// TIA Portal V16 export
// export: Created 2021-11-12T13:31:33.7596207Z, ExportSetting WithDefaults, DisplayName Totally Integrated Automation Portal, DisplayVersion V16 Update 3, DisplayName TIA Portal Version Control Interface, DisplayVersion V16 Update 2, DisplayName TIA Portal Openness, DisplayVersion V16 Update 3, DisplayName SINAMICS Startdrive Advanced, DisplayVersion V16 Update 5, DisplayName SINAMICS Startdrive G130, G150, S120, S150, SINAMICS MV, S210, DisplayVersion V16 Update 5, DisplayName SINAMICS Startdrive G110M, G120, G120C, G120D, G120P, G115D, DisplayVersion V16 Update 5, DisplayName STEP 7 Professional, DisplayVersion V16 Update 3, DisplayName STEP 7 Safety, DisplayVersion V16, DisplayName WinCC UA Professional, DisplayVersion V16 Update 3
FUNCTION_BLOCK "STD_Siemens_G120_CU240E_2_PN"   // FB1999, LAD
TITLE = Sinamics G120 with CU240E-2 PN control
{ S7_Optimized_Access := 'TRUE' }
AUTHOR : PI
FAMILY : Standard
VERSION : 0.1
// Control of Sinamics G120 with CU240E-2 PN
// 7words in/6words out (to/from PLC)
// Bi directional
// Speed and ramp control
// Errors of FI and motor evaluation
// stored: AutoNumber true, IsIECCheckEnabled false, IsRetainMemResEnabled false, MemoryReserve 100, SetENOAutomatically false, UDAEnableTagReadback false
   VAR_INPUT
      IW_HWID : HW_SUBMODULE;   // HW_Identifier - for read and write
      IB1ReqDir1 : Bool;   // Request to move in direction 1
      IB1ReqDir2 : Bool;   // Request to move in direction 2
      IB1Ack : Bool;   // Acknowledge
      IB1AlmSupp : Bool;   // Alarm suppression - external
      IB1FIProt : Bool;   // Alarm: FI Circuit Breaker / Protection of Frequency inverter OK
      IB1FICont : Bool;   // Alarm: FI Contactor / Signal from contactor on FIs input
      IB1MtrServSwch : Bool;   // Alarm: Motor 1 Service Switch / Service switch in front of motor
      IB1MtrTemp : Bool;   // Alarm: Motor 1 Thermal Protection / Temperature of motor OK
      IB1MtrBrkProt : Bool;   // Alarm: Motor 1 Brake Circuit Breaker / Protection of brake OK
      IB1MtrBrkCont : Bool;   // Alarm: Motor 1 Brake Contactor / Contactor of brake
      IB0OFF2 : Bool;   // Signal to activate OFF2 (coast)
      IB0OFF3 : Bool;   // Signal to activate OFF3 (fast ramp)
      IR_SpdSP : Real;   // Requested speed (rpm)
      IR_UpRamp { ExternalAccessible := 'False'; ExternalVisible := 'False'; ExternalWritable := 'False'} : Real := 100.0;   // Up ramp scaling 0..100%
      IR_DownRamp { ExternalAccessible := 'False'; ExternalVisible := 'False'; ExternalWritable := 'False'} : Real := 100.0;   // Down ramp scaling 0..100%
      IT_FIAlmFbk { ExternalAccessible := 'False'; ExternalVisible := 'False'; ExternalWritable := 'False'} : Time := T#100ms;   // Time to evaluate error of FI feedback
      IT_BrkAlm : Time;   // Time to evaluate error of brake release feedback
      IT_Rot : Time := T#100ms;   // Timeout for sense of rotation evaluation
   END_VAR
   VAR_OUTPUT
      OS_Status : Struct   // Output structures
         Main : "UDT_Status_main";
         Specific : "UDT_SINAMICS_G120_Status_specific";
         Error : "UDT_Error02";
      END_STRUCT;
      OW_CtrlWord1 : Word;   // Control word to FI -just for monitoring
      OB1_MtrHoldBrkOpn : Bool;   // Motor holding brake open
   END_VAR
   VAR_IN_OUT
      XS_Command : "UDT_SINAMICS_G120_Command";
      XS_Parameter : "UDT_SINAMICS_G120_Parameter";
   END_VAR
   VAR DB_SPECIFIC
      SS_Alarm : Struct   // Alarms
         FIProt : Bool;   // Frekvenční měnič - ochrana / Frequency invertor - protection / Convertisseur de fréquence - protection
         FICont : Bool;   // Frekvenční měnič - spínač / Frequency invertor - contactor / Convertisseur de fréquence - contacteur
         FIFastOff : Bool;   // Frekvenční měnič - porucha / Frequency invertor - fast off / Convertisseur de fréquence - erreur
         FIFbk : Bool;   // Frekvenční měnič - zpětná vazba chod / Frequency invertor - feedback run / Convertisseur de fréquence - rétroaction
         FITemp : Bool;   // Frekvenční měnič - vysoká teplota / Frequency invertor - high temperature / Convertisseur de fréquence - température
         FICommErr : Bool;   // Frekvenční měnič - komunikace / Frequency invertor - communication / Convertisseur de fréquence - communication
         FINotRdy : Bool;   // Frequency invertor - not ready
         Res_0_7 : Bool;   // Reserve
         MtrServSwch : Bool;   // Motor - servisní vypínač / Motor - service switch / Moteur - interrupteur de service
         MtrTemp : Bool;   // Motor - vysoká teplota / Motor - high temperature / Moteur - température
         MtrBrkProt : Bool;   // Motor - ochrana brzdy / Motor - brake protection / Moteur - protectrice de frein
         MtrBrkCont : Bool;   // Motor - spínač brzdy / Motor - brake contactor / Moteur - contacteur de frein
         MtrRot : Bool;   // Motor - sense of rotation incoherence
         Res_1_5 : Bool;   // Reserve
         Res_1_6 : Bool;   // Reserve
         InCmdIncoher : Bool;   // Dir1 and Dir2 input commands incoherence
      END_STRUCT;
      SS_Warning : Struct   // Warnings
         SpdDeviation : Bool;   // Speed deviation outside the tolerance range
         Res_0_1 : Bool;   // Reserve
         Res_0_2 : Bool;   // Reserve
         Res_0_3 : Bool;   // Reserve
         Res_0_4 : Bool;   // Reserve
         Res_0_5 : Bool;   // Reserve
         Res_0_6 : Bool;   // Reserve
         Res_0_7 : Bool;   // Reserve
         Res_1_0 : Bool;   // Reserve
         Res_1_1 : Bool;   // Reserve
         Res_1_2 : Bool;   // Reserve
         Res_1_3 : Bool;   // Reserve
         Res_1_4 : Bool;   // Reserve
         Res_1_5 : Bool;   // Reserve
         Res_1_6 : Bool;   // Reserve
         Res_1_7 : Bool;   // Reserve
      END_STRUCT;
      SI_DPRDDATRetVal { ExternalAccessible := 'False'; ExternalVisible := 'False'; ExternalWritable := 'False'} : Int;   // DPRD_DAT function return value
      SI_DPWRDATRetVal { ExternalAccessible := 'False'; ExternalVisible := 'False'; ExternalWritable := 'False'} : Int;   // DPWR_DAT function return value
      SB1DPRDWRCommOK : Bool;   // No error occurs while the instruction DPRD_DAT or DPWR_DAT is being executed
      SB1OutDir1 : Bool;   // Request to move in direction 1
      SB1OutDir2 : Bool;   // Request to move in direction 2
      ST_AlmFbk { S7_SetPoint := 'True'} : TON_TIME;   // To evaluate feedback error of FI
      ST_AlmBrake { S7_SetPoint := 'True'} : TON_TIME;   // To evaluate error on brake
      ST_AlmFIErr { S7_SetPoint := 'True'} : TON_TIME;   // To evaluate error reported from FI
   END_VAR
   VAR
      ST_RotSense { S7_SetPoint := 'True'} : TON_TIME;   // To evaluate sense of rotation incoherence
   END_VAR
   VAR DB_SPECIFIC
      ST_AckFl { S7_SetPoint := 'True'} : TP_TIME;   // TOF ack to G120
   END_VAR
   VAR_TEMP
      TS_Command : "UDT_SINAMICS_G120_Command";
      TS_Parameter : "UDT_SINAMICS_G120_Parameter";
      TS_Status : Struct
         Main : "UDT_Status_main";
         Specific : "UDT_SINAMICS_G120_Status_specific";
         Error : "UDT_Error02";
      END_STRUCT;
      TI_DPReadRet : Int;   // Result of DP reading
      TI_DPWriteRet : Int;   // Result of DP writing
      TR_Temp : Real;   // Temporary REAL value
      TS_Input : "UDT_ CU240E_I_352";   // 6 byte struct to receive data from FI
      TS_Output : "UDT_CU240E_O_352";   // 6 byte struct to send data to FI
   END_VAR
   VAR CONSTANT
      Ack : Time := T#300ms;   // Time to acknowledge FI (via PN)
   END_VAR
BEGIN

REGION Network 1: Clear temporary variables, TS_Status - Main, Specific
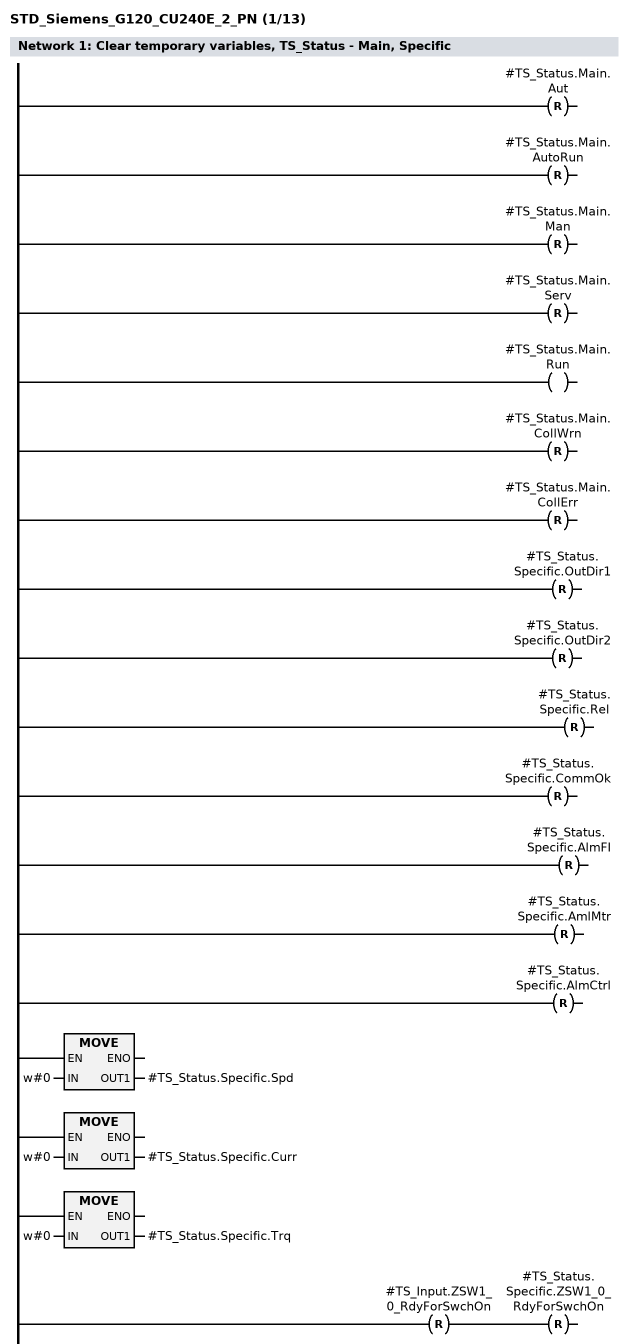
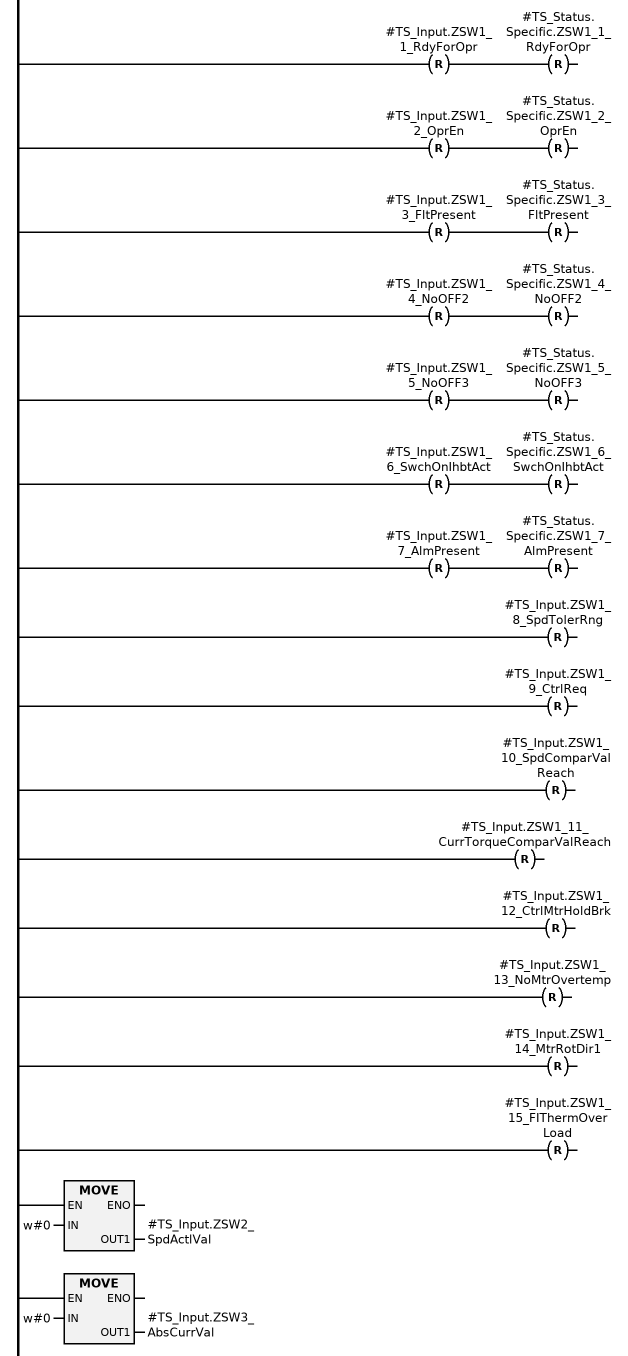
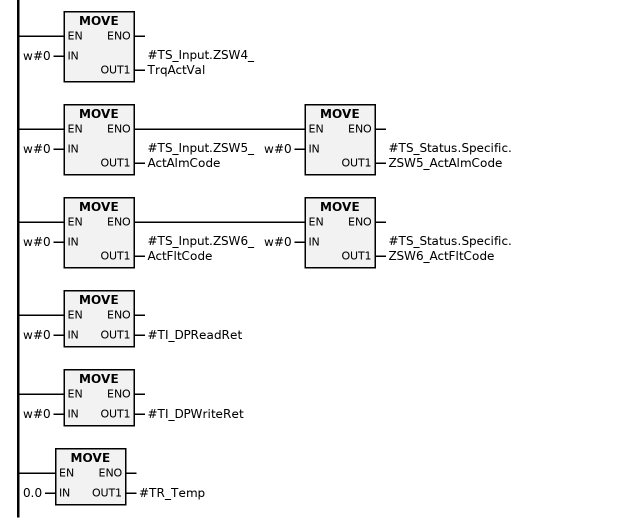
   RUNG wire#powerrail
      R_Coil( #TS_Status.Main.Aut )
   END_RUNG
   RUNG wire#powerrail
      R_Coil( #TS_Status.Main.AutoRun )
   END_RUNG
   RUNG wire#powerrail
      R_Coil( #TS_Status.Main.Man )
   END_RUNG
   RUNG wire#powerrail
      R_Coil( #TS_Status.Main.Serv )
   END_RUNG
   RUNG wire#powerrail
      Coil( #TS_Status.Main.Run )
   END_RUNG
   RUNG wire#powerrail
      R_Coil( #TS_Status.Main.CollWrn )
   END_RUNG
   RUNG wire#powerrail
      R_Coil( #TS_Status.Main.CollErr )
   END_RUNG
   RUNG wire#powerrail
      R_Coil( #TS_Status.Specific.OutDir1 )
   END_RUNG
   RUNG wire#powerrail
      R_Coil( #TS_Status.Specific.OutDir2 )
   END_RUNG
   RUNG wire#powerrail
      R_Coil( #TS_Status.Specific.Rel )
   END_RUNG
   RUNG wire#powerrail
      R_Coil( #TS_Status.Specific.CommOk )
   END_RUNG
   RUNG wire#powerrail
      R_Coil( #TS_Status.Specific.AlmFI )
   END_RUNG
   RUNG wire#powerrail
      R_Coil( #TS_Status.Specific.AmlMtr )
   END_RUNG
   RUNG wire#powerrail
      R_Coil( #TS_Status.Specific.AlmCtrl )
   END_RUNG
   RUNG wire#powerrail
      { S7_GenerateENO := "TRUE" } Move(in := w#0, out1 => #TS_Status.Specific.Spd)
   END_RUNG
   RUNG wire#powerrail
      { S7_GenerateENO := "TRUE" } Move(in := w#0, out1 => #TS_Status.Specific.Curr)
   END_RUNG
   RUNG wire#powerrail
      { S7_GenerateENO := "TRUE" } Move(in := w#0, out1 => #TS_Status.Specific.Trq)
   END_RUNG
   RUNG wire#powerrail
      R_Coil( #TS_Input.ZSW1_0_RdyForSwchOn )
      R_Coil( #TS_Status.Specific.ZSW1_0_RdyForSwchOn )
   END_RUNG
   RUNG wire#powerrail
      R_Coil( #TS_Input.ZSW1_1_RdyForOpr )
      R_Coil( #TS_Status.Specific.ZSW1_1_RdyForOpr )
   END_RUNG
   RUNG wire#powerrail
      R_Coil( #TS_Input.ZSW1_2_OprEn )
      R_Coil( #TS_Status.Specific.ZSW1_2_OprEn )
   END_RUNG
   RUNG wire#powerrail
      R_Coil( #TS_Input.ZSW1_3_FltPresent )
      R_Coil( #TS_Status.Specific.ZSW1_3_FltPresent )
   END_RUNG
   RUNG wire#powerrail
      R_Coil( #TS_Input.ZSW1_4_NoOFF2 )
      R_Coil( #TS_Status.Specific.ZSW1_4_NoOFF2 )
   END_RUNG
   RUNG wire#powerrail
      R_Coil( #TS_Input.ZSW1_5_NoOFF3 )
      R_Coil( #TS_Status.Specific.ZSW1_5_NoOFF3 )
   END_RUNG
   RUNG wire#powerrail
      R_Coil( #TS_Input.ZSW1_6_SwchOnIhbtAct )
      R_Coil( #TS_Status.Specific.ZSW1_6_SwchOnIhbtAct )
   END_RUNG
   RUNG wire#powerrail
      R_Coil( #TS_Input.ZSW1_7_AlmPresent )
      R_Coil( #TS_Status.Specific.ZSW1_7_AlmPresent )
   END_RUNG
   RUNG wire#powerrail
      R_Coil( #TS_Input.ZSW1_8_SpdTolerRng )
   END_RUNG
   RUNG wire#powerrail
      R_Coil( #TS_Input.ZSW1_9_CtrlReq )
   END_RUNG
   RUNG wire#powerrail
      R_Coil( #TS_Input.ZSW1_10_SpdComparValReach )
   END_RUNG
   RUNG wire#powerrail
      R_Coil( #TS_Input.ZSW1_11_CurrTorqueComparValReach )
   END_RUNG
   RUNG wire#powerrail
      R_Coil( #TS_Input.ZSW1_12_CtrlMtrHoldBrk )
   END_RUNG
   RUNG wire#powerrail
      R_Coil( #TS_Input.ZSW1_13_NoMtrOvertemp )
   END_RUNG
   RUNG wire#powerrail
      R_Coil( #TS_Input.ZSW1_14_MtrRotDir1 )
   END_RUNG
   RUNG wire#powerrail
      R_Coil( #TS_Input.ZSW1_15_FIThermOverLoad )
   END_RUNG
   RUNG wire#powerrail
      { S7_GenerateENO := "TRUE" } Move(in := w#0, out1 => #TS_Input.ZSW2_SpdActlVal)
   END_RUNG
   RUNG wire#powerrail
      { S7_GenerateENO := "TRUE" } Move(in := w#0, out1 => #TS_Input.ZSW3_AbsCurrVal)
   END_RUNG
   RUNG wire#powerrail
      { S7_GenerateENO := "TRUE" } Move(in := w#0, out1 => #TS_Input.ZSW4_TrqActVal)
   END_RUNG
   RUNG wire#powerrail
      { S7_GenerateENO := "TRUE" } Move(in := w#0, out1 => #TS_Input.ZSW5_ActAlmCode)
      { S7_GenerateENO := "TRUE" } Move(in := w#0, out1 => #TS_Status.Specific.ZSW5_ActAlmCode)
   END_RUNG
   RUNG wire#powerrail
      { S7_GenerateENO := "TRUE" } Move(in := w#0, out1 => #TS_Input.ZSW6_ActFltCode)
      { S7_GenerateENO := "TRUE" } Move(in := w#0, out1 => #TS_Status.Specific.ZSW6_ActFltCode)
   END_RUNG
   RUNG wire#powerrail
      { S7_GenerateENO := "TRUE" } Move(in := w#0, out1 => #TI_DPReadRet)
   END_RUNG
   RUNG wire#powerrail
      { S7_GenerateENO := "TRUE" } Move(in := w#0, out1 => #TI_DPWriteRet)
   END_RUNG
   RUNG wire#powerrail
      { S7_GenerateENO := "TRUE" } Move(in := 0.0, out1 => #TR_Temp)
   END_RUNG
   // the same network as SCL:
   // ENO of a box is taken as its EN; it also drops when the box reports an error
   #TS_Status.Main.Aut := FALSE;
   #TS_Status.Main.AutoRun := FALSE;
   #TS_Status.Main.Man := FALSE;
   #TS_Status.Main.Serv := FALSE;
   #TS_Status.Main.Run := TRUE;
   #TS_Status.Main.CollWrn := FALSE;
   #TS_Status.Main.CollErr := FALSE;
   #TS_Status.Specific.OutDir1 := FALSE;
   #TS_Status.Specific.OutDir2 := FALSE;
   #TS_Status.Specific.Rel := FALSE;
   #TS_Status.Specific.CommOk := FALSE;
   #TS_Status.Specific.AlmFI := FALSE;
   #TS_Status.Specific.AmlMtr := FALSE;
   #TS_Status.Specific.AlmCtrl := FALSE;
   #TS_Status.Specific.Spd := w#0;
   #TS_Status.Specific.Curr := w#0;
   #TS_Status.Specific.Trq := w#0;
   #TS_Input.ZSW1_0_RdyForSwchOn := FALSE;
   #TS_Status.Specific.ZSW1_0_RdyForSwchOn := FALSE;
   #TS_Input.ZSW1_1_RdyForOpr := FALSE;
   #TS_Status.Specific.ZSW1_1_RdyForOpr := FALSE;
   #TS_Input.ZSW1_2_OprEn := FALSE;
   #TS_Status.Specific.ZSW1_2_OprEn := FALSE;
   #TS_Input.ZSW1_3_FltPresent := FALSE;
   #TS_Status.Specific.ZSW1_3_FltPresent := FALSE;
   #TS_Input.ZSW1_4_NoOFF2 := FALSE;
   #TS_Status.Specific.ZSW1_4_NoOFF2 := FALSE;
   #TS_Input.ZSW1_5_NoOFF3 := FALSE;
   #TS_Status.Specific.ZSW1_5_NoOFF3 := FALSE;
   #TS_Input.ZSW1_6_SwchOnIhbtAct := FALSE;
   #TS_Status.Specific.ZSW1_6_SwchOnIhbtAct := FALSE;
   #TS_Input.ZSW1_7_AlmPresent := FALSE;
   #TS_Status.Specific.ZSW1_7_AlmPresent := FALSE;
   #TS_Input.ZSW1_8_SpdTolerRng := FALSE;
   #TS_Input.ZSW1_9_CtrlReq := FALSE;
   #TS_Input.ZSW1_10_SpdComparValReach := FALSE;
   #TS_Input.ZSW1_11_CurrTorqueComparValReach := FALSE;
   #TS_Input.ZSW1_12_CtrlMtrHoldBrk := FALSE;
   #TS_Input.ZSW1_13_NoMtrOvertemp := FALSE;
   #TS_Input.ZSW1_14_MtrRotDir1 := FALSE;
   #TS_Input.ZSW1_15_FIThermOverLoad := FALSE;
   #TS_Input.ZSW2_SpdActlVal := w#0;
   #TS_Input.ZSW3_AbsCurrVal := w#0;
   #TS_Input.ZSW4_TrqActVal := w#0;
   #TS_Input.ZSW5_ActAlmCode := w#0;
   #TS_Status.Specific.ZSW5_ActAlmCode := w#0;
   #TS_Input.ZSW6_ActFltCode := w#0;
   #TS_Status.Specific.ZSW6_ActFltCode := w#0;
   #TI_DPReadRet := w#0;
   #TI_DPWriteRet := w#0;
   #TR_Temp := 0.0;
END_REGION

REGION Network 2: Copy In/Out variables into temporary variables
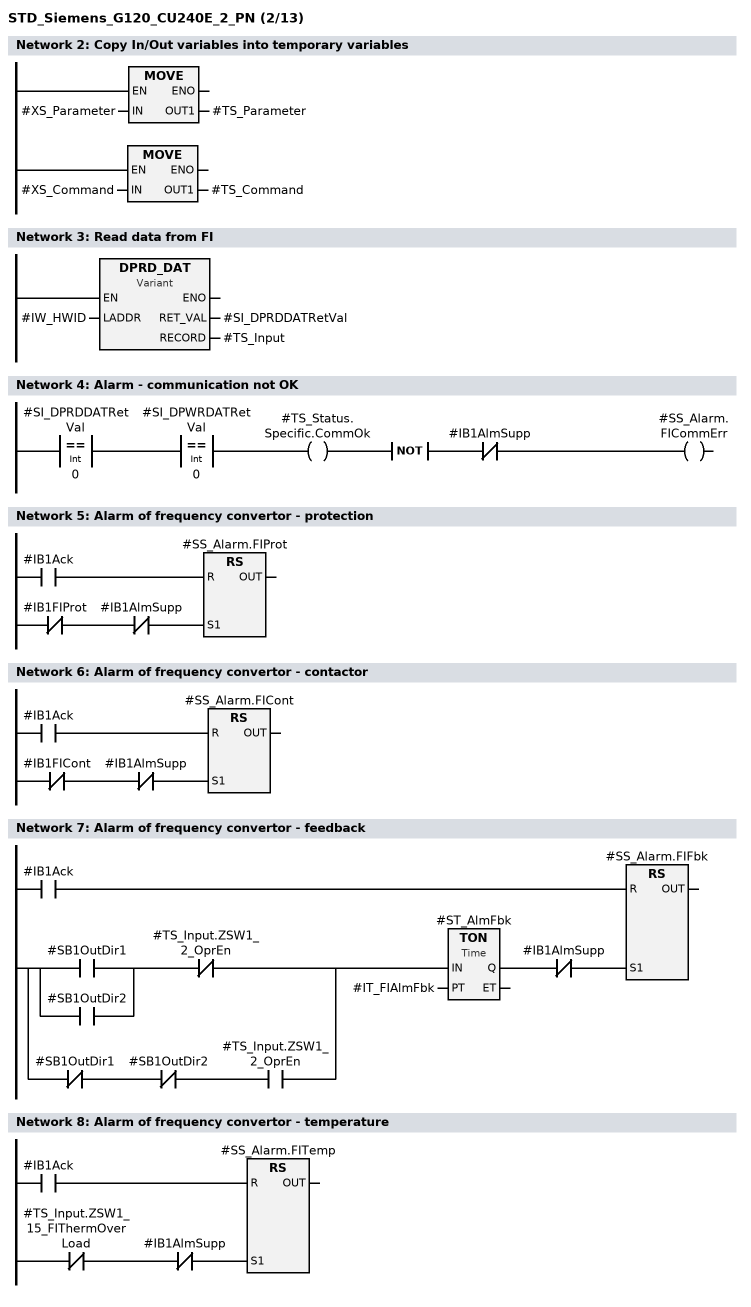
   RUNG wire#powerrail
      { S7_GenerateENO := "TRUE" } Move(in := #XS_Parameter, out1 => #TS_Parameter)
   END_RUNG
   RUNG wire#powerrail
      { S7_GenerateENO := "TRUE" } Move(in := #XS_Command, out1 => #TS_Command)
   END_RUNG
   // the same network as SCL:
   #TS_Parameter := #XS_Parameter;
   #TS_Command := #XS_Command;
END_REGION

REGION Network 3: Read data from FI
   RUNG wire#powerrail
      { S7_Templates := "[ptr_type := Variant, laddr_type := HW_IO]" } DPRD_DAT(LADDR := #IW_HWID, RET_VAL => #SI_DPRDDATRetVal, RECORD => #TS_Input)
   END_RUNG
   // the same network as SCL:
   #SI_DPRDDATRetVal := DPRD_DAT(LADDR := #IW_HWID, RECORD => #TS_Input);
END_REGION

REGION Network 4: Alarm - communication not OK
   RUNG wire#powerrail
      { S7_Templates := "SrcType := Int" } EQ_Contact(in1 := #SI_DPRDDATRetVal, in2 := 0)
      { S7_Templates := "SrcType := Int" } EQ_Contact(in1 := #SI_DPWRDATRetVal, in2 := 0)
      Coil( #TS_Status.Specific.CommOk )
      Not()
      I_Contact( #IB1AlmSupp )
      Coil( #SS_Alarm.FICommErr )
   END_RUNG
   // the same network as SCL:
   #TS_Status.Specific.CommOk := (#SI_DPRDDATRetVal = 0) AND (#SI_DPWRDATRetVal = 0);
   #SS_Alarm.FICommErr := NOT #TS_Status.Specific.CommOk AND NOT #IB1AlmSupp;
END_REGION

REGION Network 5: Alarm of frequency convertor - protection
   RUNG wire#powerrail
      Contact( #IB1Ack )
      S_RS(operand := #SS_Alarm.FIProt, s1 := wire#w1)
   END_RUNG
   RUNG wire#powerrail
      I_Contact( #IB1FIProt )
      I_Contact( #IB1AlmSupp )
   END_RUNG wire#w1
   // the same network as SCL:
   IF #IB1Ack THEN
       #SS_Alarm.FIProt := FALSE;   // RS flip-flop
   END_IF;
   IF NOT #IB1FIProt AND NOT #IB1AlmSupp THEN #SS_Alarm.FIProt := TRUE; END_IF;
END_REGION

REGION Network 6: Alarm of frequency convertor - contactor
   RUNG wire#powerrail
      Contact( #IB1Ack )
      S_RS(operand := #SS_Alarm.FICont, s1 := wire#w1)
   END_RUNG
   RUNG wire#powerrail
      I_Contact( #IB1FICont )
      I_Contact( #IB1AlmSupp )
   END_RUNG wire#w1
   // the same network as SCL:
   IF #IB1Ack THEN
       #SS_Alarm.FICont := FALSE;   // RS flip-flop
   END_IF;
   IF NOT #IB1FICont AND NOT #IB1AlmSupp THEN #SS_Alarm.FICont := TRUE; END_IF;
END_REGION

REGION Network 7: Alarm of frequency convertor - feedback
   RUNG wire#powerrail
      Contact( #IB1Ack )
      S_RS(operand := #SS_Alarm.FIFbk, s1 := wire#w3)
   END_RUNG
   RUNG wire#powerrail
      Contact( #SB1OutDir1 )
      wire#w1
      I_Contact( #TS_Input.ZSW1_2_OprEn )
      wire#w2
      { S7_Templates := "time_type := Time" } #ST_AlmFbk.TON(pt := #IT_FIAlmFbk, et =>)
      I_Contact( #IB1AlmSupp )
   END_RUNG wire#w3
   RUNG wire#powerrail
      Contact( #SB1OutDir2 )
   END_RUNG wire#w1
   RUNG wire#powerrail
      I_Contact( #SB1OutDir1 )
      I_Contact( #SB1OutDir2 )
      Contact( #TS_Input.ZSW1_2_OprEn )
   END_RUNG wire#w2
   // the same network as SCL:
   #ST_AlmFbk(IN := ((#SB1OutDir1 OR #SB1OutDir2) AND NOT #TS_Input.ZSW1_2_OprEn) OR (NOT #SB1OutDir1 AND NOT #SB1OutDir2 AND #TS_Input.ZSW1_2_OprEn),   // TON
              PT := #IT_FIAlmFbk);
   IF #IB1Ack THEN
       #SS_Alarm.FIFbk := FALSE;   // RS flip-flop
   END_IF;
   IF #ST_AlmFbk.Q AND NOT #IB1AlmSupp THEN #SS_Alarm.FIFbk := TRUE; END_IF;
END_REGION

REGION Network 8: Alarm of frequency convertor - temperature
   RUNG wire#powerrail
      Contact( #IB1Ack )
      S_RS(operand := #SS_Alarm.FITemp, s1 := wire#w1)
   END_RUNG
   RUNG wire#powerrail
      I_Contact( #TS_Input.ZSW1_15_FIThermOverLoad )
      I_Contact( #IB1AlmSupp )
   END_RUNG wire#w1
   // the same network as SCL:
   IF #IB1Ack THEN
       #SS_Alarm.FITemp := FALSE;   // RS flip-flop
   END_IF;
   IF NOT #TS_Input.ZSW1_15_FIThermOverLoad AND NOT #IB1AlmSupp THEN #SS_Alarm.FITemp := TRUE; END_IF;
END_REGION

REGION Network 9: Alarm of motor - service switch off
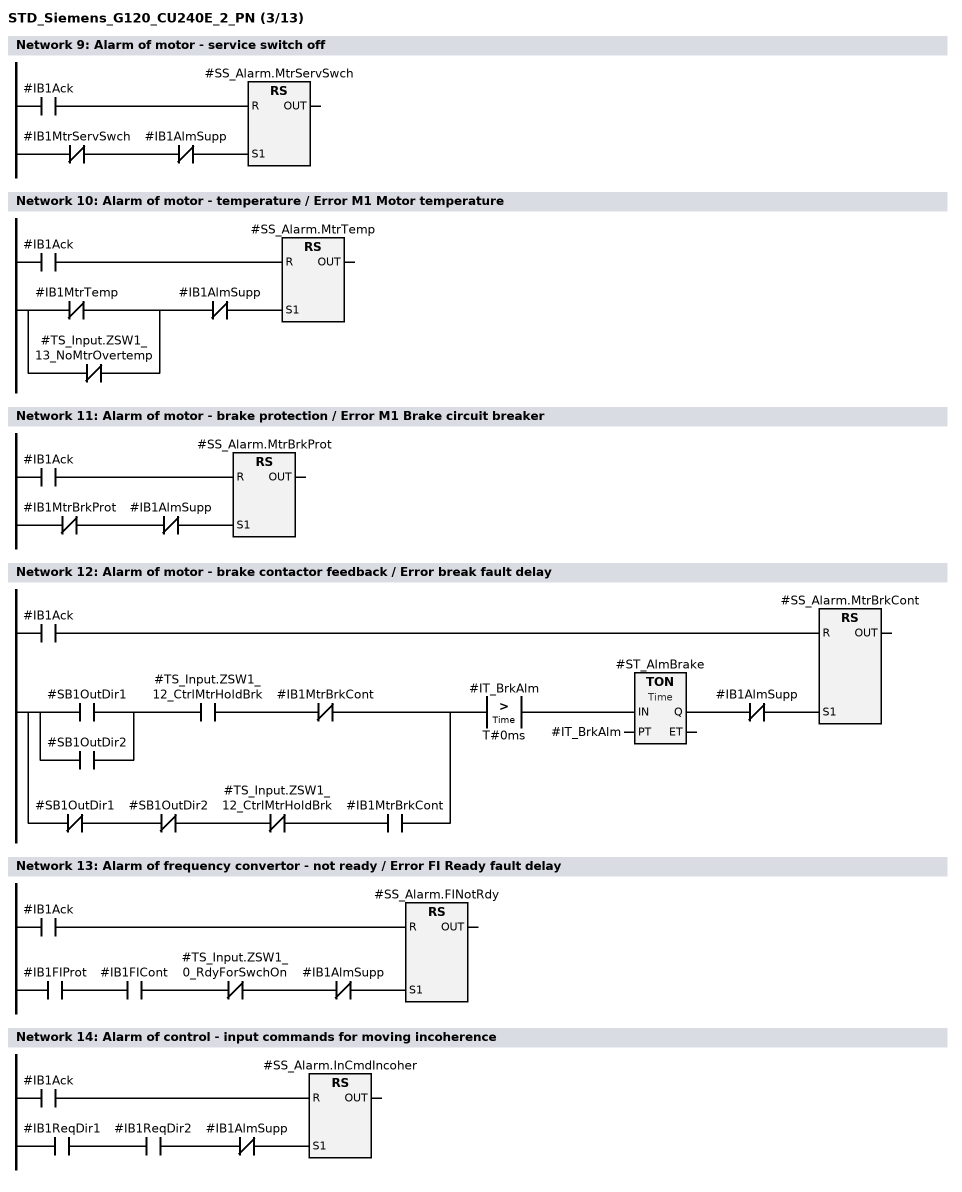
   RUNG wire#powerrail
      Contact( #IB1Ack )
      S_RS(operand := #SS_Alarm.MtrServSwch, s1 := wire#w1)
   END_RUNG
   RUNG wire#powerrail
      I_Contact( #IB1MtrServSwch )
      I_Contact( #IB1AlmSupp )
   END_RUNG wire#w1
   // the same network as SCL:
   IF #IB1Ack THEN
       #SS_Alarm.MtrServSwch := FALSE;   // RS flip-flop
   END_IF;
   IF NOT #IB1MtrServSwch AND NOT #IB1AlmSupp THEN #SS_Alarm.MtrServSwch := TRUE; END_IF;
END_REGION

REGION Network 10: Alarm of motor - temperature / Error M1 Motor temperature
   RUNG wire#powerrail
      Contact( #IB1Ack )
      S_RS(operand := #SS_Alarm.MtrTemp, s1 := wire#w2)
   END_RUNG
   RUNG wire#powerrail
      I_Contact( #IB1MtrTemp )
      wire#w1
      I_Contact( #IB1AlmSupp )
   END_RUNG wire#w2
   RUNG wire#powerrail
      I_Contact( #TS_Input.ZSW1_13_NoMtrOvertemp )
   END_RUNG wire#w1
   // the same network as SCL:
   IF #IB1Ack THEN
       #SS_Alarm.MtrTemp := FALSE;   // RS flip-flop
   END_IF;
   IF (NOT #IB1MtrTemp OR NOT #TS_Input.ZSW1_13_NoMtrOvertemp) AND NOT #IB1AlmSupp THEN
       #SS_Alarm.MtrTemp := TRUE;
   END_IF;
END_REGION

REGION Network 11: Alarm of motor - brake protection / Error M1 Brake circuit breaker
   RUNG wire#powerrail
      Contact( #IB1Ack )
      S_RS(operand := #SS_Alarm.MtrBrkProt, s1 := wire#w1)
   END_RUNG
   RUNG wire#powerrail
      I_Contact( #IB1MtrBrkProt )
      I_Contact( #IB1AlmSupp )
   END_RUNG wire#w1
   // the same network as SCL:
   IF #IB1Ack THEN
       #SS_Alarm.MtrBrkProt := FALSE;   // RS flip-flop
   END_IF;
   IF NOT #IB1MtrBrkProt AND NOT #IB1AlmSupp THEN #SS_Alarm.MtrBrkProt := TRUE; END_IF;
END_REGION

REGION Network 12: Alarm of motor - brake contactor feedback / Error break fault delay
   RUNG wire#powerrail
      Contact( #IB1Ack )
      S_RS(operand := #SS_Alarm.MtrBrkCont, s1 := wire#w3)
   END_RUNG
   RUNG wire#powerrail
      Contact( #SB1OutDir1 )
      wire#w1
      Contact( #TS_Input.ZSW1_12_CtrlMtrHoldBrk )
      I_Contact( #IB1MtrBrkCont )
      wire#w2
      { S7_Templates := "SrcType := Time" } GT_Contact(in1 := #IT_BrkAlm, in2 := T#0ms)
      { S7_Templates := "time_type := Time" } #ST_AlmBrake.TON(pt := #IT_BrkAlm, et =>)
      I_Contact( #IB1AlmSupp )
   END_RUNG wire#w3
   RUNG wire#powerrail
      Contact( #SB1OutDir2 )
   END_RUNG wire#w1
   RUNG wire#powerrail
      I_Contact( #SB1OutDir1 )
      I_Contact( #SB1OutDir2 )
      I_Contact( #TS_Input.ZSW1_12_CtrlMtrHoldBrk )
      Contact( #IB1MtrBrkCont )
   END_RUNG wire#w2
   // the same network as SCL:
   #ST_AlmBrake(IN := (((#SB1OutDir1 OR #SB1OutDir2) AND #TS_Input.ZSW1_12_CtrlMtrHoldBrk AND NOT #IB1MtrBrkCont) OR (NOT #SB1OutDir1 AND NOT #SB1OutDir2 AND NOT #TS_Input.ZSW1_12_CtrlMtrHoldBrk AND #IB1MtrBrkCont)) AND (#IT_BrkAlm > T#0ms),   // TON
                PT := #IT_BrkAlm);
   IF #IB1Ack THEN
       #SS_Alarm.MtrBrkCont := FALSE;   // RS flip-flop
   END_IF;
   IF #ST_AlmBrake.Q AND NOT #IB1AlmSupp THEN #SS_Alarm.MtrBrkCont := TRUE; END_IF;
END_REGION

REGION Network 13: Alarm of frequency convertor - not ready / Error FI Ready fault delay
   RUNG wire#powerrail
      Contact( #IB1Ack )
      S_RS(operand := #SS_Alarm.FINotRdy, s1 := wire#w1)
   END_RUNG
   RUNG wire#powerrail
      Contact( #IB1FIProt )
      Contact( #IB1FICont )
      I_Contact( #TS_Input.ZSW1_0_RdyForSwchOn )
      I_Contact( #IB1AlmSupp )
   END_RUNG wire#w1
   // the same network as SCL:
   IF #IB1Ack THEN
       #SS_Alarm.FINotRdy := FALSE;   // RS flip-flop
   END_IF;
   IF #IB1FIProt AND #IB1FICont AND NOT #TS_Input.ZSW1_0_RdyForSwchOn AND NOT #IB1AlmSupp THEN
       #SS_Alarm.FINotRdy := TRUE;
   END_IF;
END_REGION

REGION Network 14: Alarm of control - input commands for moving incoherence
   RUNG wire#powerrail
      Contact( #IB1Ack )
      S_RS(operand := #SS_Alarm.InCmdIncoher, s1 := wire#w1)
   END_RUNG
   RUNG wire#powerrail
      Contact( #IB1ReqDir1 )
      Contact( #IB1ReqDir2 )
      I_Contact( #IB1AlmSupp )
   END_RUNG wire#w1
   // the same network as SCL:
   IF #IB1Ack THEN
       #SS_Alarm.InCmdIncoher := FALSE;   // RS flip-flop
   END_IF;
   IF #IB1ReqDir1 AND #IB1ReqDir2 AND NOT #IB1AlmSupp THEN #SS_Alarm.InCmdIncoher := TRUE; END_IF;
END_REGION

REGION Network 15: Alarm of motor - sense of rotation incoherence
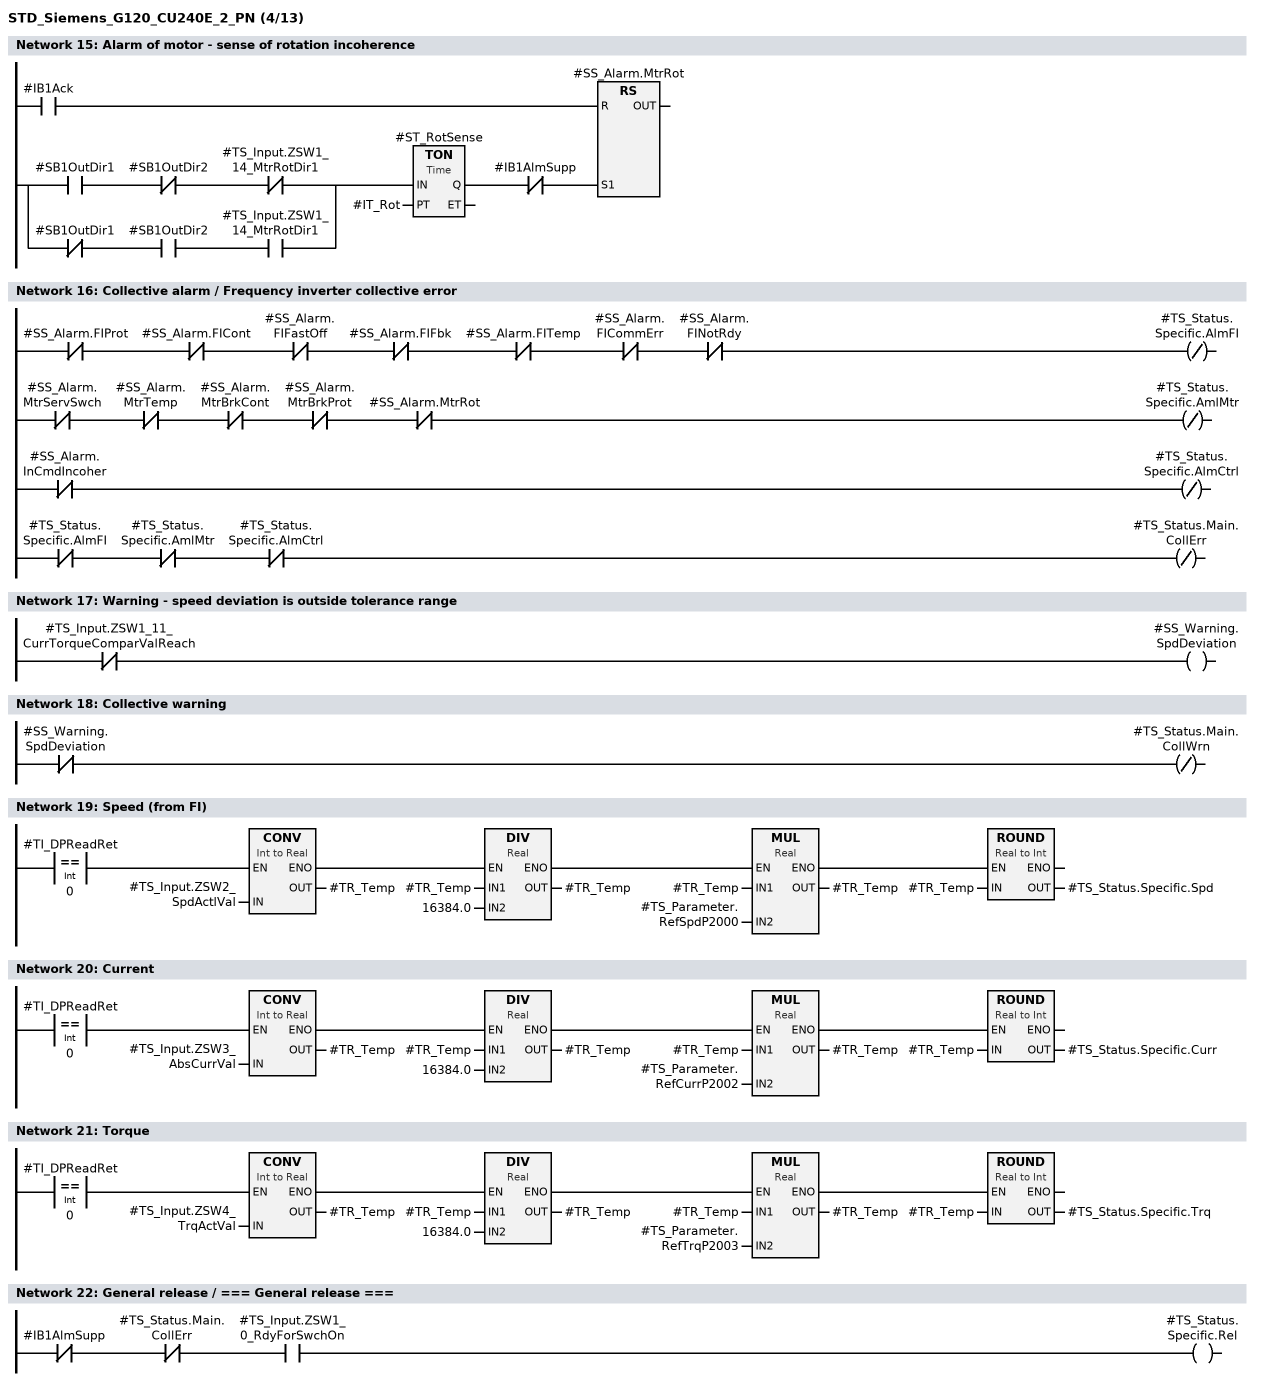
   RUNG wire#powerrail
      Contact( #IB1Ack )
      S_RS(operand := #SS_Alarm.MtrRot, s1 := wire#w2)
   END_RUNG
   RUNG wire#powerrail
      Contact( #SB1OutDir1 )
      I_Contact( #SB1OutDir2 )
      I_Contact( #TS_Input.ZSW1_14_MtrRotDir1 )
      wire#w1
      { S7_Templates := "time_type := Time" } #ST_RotSense.TON(pt := #IT_Rot, et =>)
      I_Contact( #IB1AlmSupp )
   END_RUNG wire#w2
   RUNG wire#powerrail
      I_Contact( #SB1OutDir1 )
      Contact( #SB1OutDir2 )
      Contact( #TS_Input.ZSW1_14_MtrRotDir1 )
   END_RUNG wire#w1
   // the same network as SCL:
   #ST_RotSense(IN := (#SB1OutDir1 AND NOT #SB1OutDir2 AND NOT #TS_Input.ZSW1_14_MtrRotDir1) OR (NOT #SB1OutDir1 AND #SB1OutDir2 AND #TS_Input.ZSW1_14_MtrRotDir1),   // TON
                PT := #IT_Rot);
   IF #IB1Ack THEN
       #SS_Alarm.MtrRot := FALSE;   // RS flip-flop
   END_IF;
   IF #ST_RotSense.Q AND NOT #IB1AlmSupp THEN #SS_Alarm.MtrRot := TRUE; END_IF;
END_REGION

REGION Network 16: Collective alarm / Frequency inverter collective error
   RUNG wire#powerrail
      I_Contact( #SS_Alarm.FIProt )
      I_Contact( #SS_Alarm.FICont )
      I_Contact( #SS_Alarm.FIFastOff )
      I_Contact( #SS_Alarm.FIFbk )
      I_Contact( #SS_Alarm.FITemp )
      I_Contact( #SS_Alarm.FICommErr )
      I_Contact( #SS_Alarm.FINotRdy )
      I_Coil( #TS_Status.Specific.AlmFI )
   END_RUNG
   RUNG wire#powerrail
      I_Contact( #SS_Alarm.MtrServSwch )
      I_Contact( #SS_Alarm.MtrTemp )
      I_Contact( #SS_Alarm.MtrBrkCont )
      I_Contact( #SS_Alarm.MtrBrkProt )
      I_Contact( #SS_Alarm.MtrRot )
      I_Coil( #TS_Status.Specific.AmlMtr )
   END_RUNG
   RUNG wire#powerrail
      I_Contact( #SS_Alarm.InCmdIncoher )
      I_Coil( #TS_Status.Specific.AlmCtrl )
   END_RUNG
   RUNG wire#powerrail
      I_Contact( #TS_Status.Specific.AlmFI )
      I_Contact( #TS_Status.Specific.AmlMtr )
      I_Contact( #TS_Status.Specific.AlmCtrl )
      I_Coil( #TS_Status.Main.CollErr )
   END_RUNG
   // the same network as SCL:
   #TS_Status.Specific.AlmFI := NOT (NOT #SS_Alarm.FIProt AND NOT #SS_Alarm.FICont AND NOT #SS_Alarm.FIFastOff AND NOT #SS_Alarm.FIFbk AND NOT #SS_Alarm.FITemp AND NOT #SS_Alarm.FICommErr AND NOT #SS_Alarm.FINotRdy);
   #TS_Status.Specific.AmlMtr := NOT (NOT #SS_Alarm.MtrServSwch AND NOT #SS_Alarm.MtrTemp AND NOT #SS_Alarm.MtrBrkCont AND NOT #SS_Alarm.MtrBrkProt AND NOT #SS_Alarm.MtrRot);
   #TS_Status.Specific.AlmCtrl := NOT (NOT #SS_Alarm.InCmdIncoher);
   #TS_Status.Main.CollErr := NOT (NOT #TS_Status.Specific.AlmFI AND NOT #TS_Status.Specific.AmlMtr AND NOT #TS_Status.Specific.AlmCtrl);
END_REGION

REGION Network 17: Warning - speed deviation is outside tolerance range
   RUNG wire#powerrail
      I_Contact( #TS_Input.ZSW1_11_CurrTorqueComparValReach )
      Coil( #SS_Warning.SpdDeviation )
   END_RUNG
   // the same network as SCL:
   #SS_Warning.SpdDeviation := NOT #TS_Input.ZSW1_11_CurrTorqueComparValReach;
END_REGION

REGION Network 18: Collective warning
   RUNG wire#powerrail
      I_Contact( #SS_Warning.SpdDeviation )
      I_Coil( #TS_Status.Main.CollWrn )
   END_RUNG
   // the same network as SCL:
   #TS_Status.Main.CollWrn := NOT (NOT #SS_Warning.SpdDeviation);
END_REGION

REGION Network 19: Speed (from FI)
   RUNG wire#powerrail
      { S7_Templates := "SrcType := Int" } EQ_Contact(in1 := #TI_DPReadRet, in2 := 0)
      { S7_Templates := "[SrcType := Int, DestType := Real]"; S7_GenerateENO := "TRUE" } Convert(in := #TS_Input.ZSW2_SpdActlVal, out => #TR_Temp)
      { S7_Templates := "SrcType := Real"; S7_GenerateENO := "TRUE" } Div(in1 := #TR_Temp, in2 := 16384.0, out => #TR_Temp)
      { S7_Templates := "SrcType := Real"; S7_GenerateENO := "TRUE" } Mul(in1 := #TR_Temp, in2 := #TS_Parameter.RefSpdP2000, out => #TR_Temp)
      { S7_Templates := "[SrcType := Real, DestType := Int]"; S7_GenerateENO := "TRUE" } Round(in := #TR_Temp, out => #TS_Status.Specific.Spd)
   END_RUNG
   // the same network as SCL:
   // ENO of a box is taken as its EN; it also drops when the box reports an error
   IF #TI_DPReadRet = 0 THEN
       #TR_Temp := INT_TO_REAL(#TS_Input.ZSW2_SpdActlVal);
       #TR_Temp := #TR_Temp / 16384.0;
       #TR_Temp := #TR_Temp * #TS_Parameter.RefSpdP2000;
       #TS_Status.Specific.Spd := ROUND(#TR_Temp);
   END_IF;
END_REGION

REGION Network 20: Current
   RUNG wire#powerrail
      { S7_Templates := "SrcType := Int" } EQ_Contact(in1 := #TI_DPReadRet, in2 := 0)
      { S7_Templates := "[SrcType := Int, DestType := Real]"; S7_GenerateENO := "TRUE" } Convert(in := #TS_Input.ZSW3_AbsCurrVal, out => #TR_Temp)
      { S7_Templates := "SrcType := Real"; S7_GenerateENO := "TRUE" } Div(in1 := #TR_Temp, in2 := 16384.0, out => #TR_Temp)
      { S7_Templates := "SrcType := Real"; S7_GenerateENO := "TRUE" } Mul(in1 := #TR_Temp, in2 := #TS_Parameter.RefCurrP2002, out => #TR_Temp)
      { S7_Templates := "[SrcType := Real, DestType := Int]"; S7_GenerateENO := "TRUE" } Round(in := #TR_Temp, out => #TS_Status.Specific.Curr)
   END_RUNG
   // the same network as SCL:
   // ENO of a box is taken as its EN; it also drops when the box reports an error
   IF #TI_DPReadRet = 0 THEN
       #TR_Temp := INT_TO_REAL(#TS_Input.ZSW3_AbsCurrVal);
       #TR_Temp := #TR_Temp / 16384.0;
       #TR_Temp := #TR_Temp * #TS_Parameter.RefCurrP2002;
       #TS_Status.Specific.Curr := ROUND(#TR_Temp);
   END_IF;
END_REGION

REGION Network 21: Torque
   RUNG wire#powerrail
      { S7_Templates := "SrcType := Int" } EQ_Contact(in1 := #TI_DPReadRet, in2 := 0)
      { S7_Templates := "[SrcType := Int, DestType := Real]"; S7_GenerateENO := "TRUE" } Convert(in := #TS_Input.ZSW4_TrqActVal, out => #TR_Temp)
      { S7_Templates := "SrcType := Real"; S7_GenerateENO := "TRUE" } Div(in1 := #TR_Temp, in2 := 16384.0, out => #TR_Temp)
      { S7_Templates := "SrcType := Real"; S7_GenerateENO := "TRUE" } Mul(in1 := #TR_Temp, in2 := #TS_Parameter.RefTrqP2003, out => #TR_Temp)
      { S7_Templates := "[SrcType := Real, DestType := Int]"; S7_GenerateENO := "TRUE" } Round(in := #TR_Temp, out => #TS_Status.Specific.Trq)
   END_RUNG
   // the same network as SCL:
   // ENO of a box is taken as its EN; it also drops when the box reports an error
   IF #TI_DPReadRet = 0 THEN
       #TR_Temp := INT_TO_REAL(#TS_Input.ZSW4_TrqActVal);
       #TR_Temp := #TR_Temp / 16384.0;
       #TR_Temp := #TR_Temp * #TS_Parameter.RefTrqP2003;
       #TS_Status.Specific.Trq := ROUND(#TR_Temp);
   END_IF;
END_REGION

REGION Network 22: General release / === General release ===
   RUNG wire#powerrail
      I_Contact( #IB1AlmSupp )
      I_Contact( #TS_Status.Main.CollErr )
      Contact( #TS_Input.ZSW1_0_RdyForSwchOn )
      Coil( #TS_Status.Specific.Rel )
   END_RUNG
   // the same network as SCL:
   #TS_Status.Specific.Rel := NOT #IB1AlmSupp AND NOT #TS_Status.Main.CollErr AND #TS_Input.ZSW1_0_RdyForSwchOn;
END_REGION

REGION Network 23: Out direction 1 / Output Forward
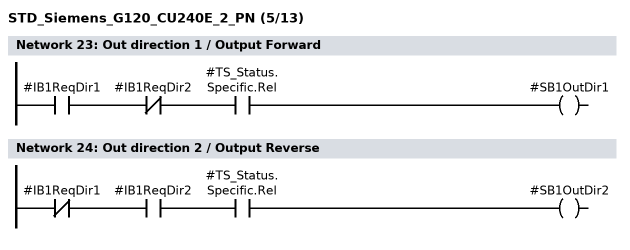
   RUNG wire#powerrail
      Contact( #IB1ReqDir1 )
      I_Contact( #IB1ReqDir2 )
      Contact( #TS_Status.Specific.Rel )
      Coil( #SB1OutDir1 )
   END_RUNG
   // the same network as SCL:
   #SB1OutDir1 := #IB1ReqDir1 AND NOT #IB1ReqDir2 AND #TS_Status.Specific.Rel;
END_REGION

REGION Network 24: Out direction 2 / Output Reverse
   RUNG wire#powerrail
      I_Contact( #IB1ReqDir1 )
      Contact( #IB1ReqDir2 )
      Contact( #TS_Status.Specific.Rel )
      Coil( #SB1OutDir2 )
   END_RUNG
   // the same network as SCL:
   #SB1OutDir2 := NOT #IB1ReqDir1 AND #IB1ReqDir2 AND #TS_Status.Specific.Rel;
END_REGION

REGION Network 25: Control word 1 - FI commands / === OS_ControlWord ===
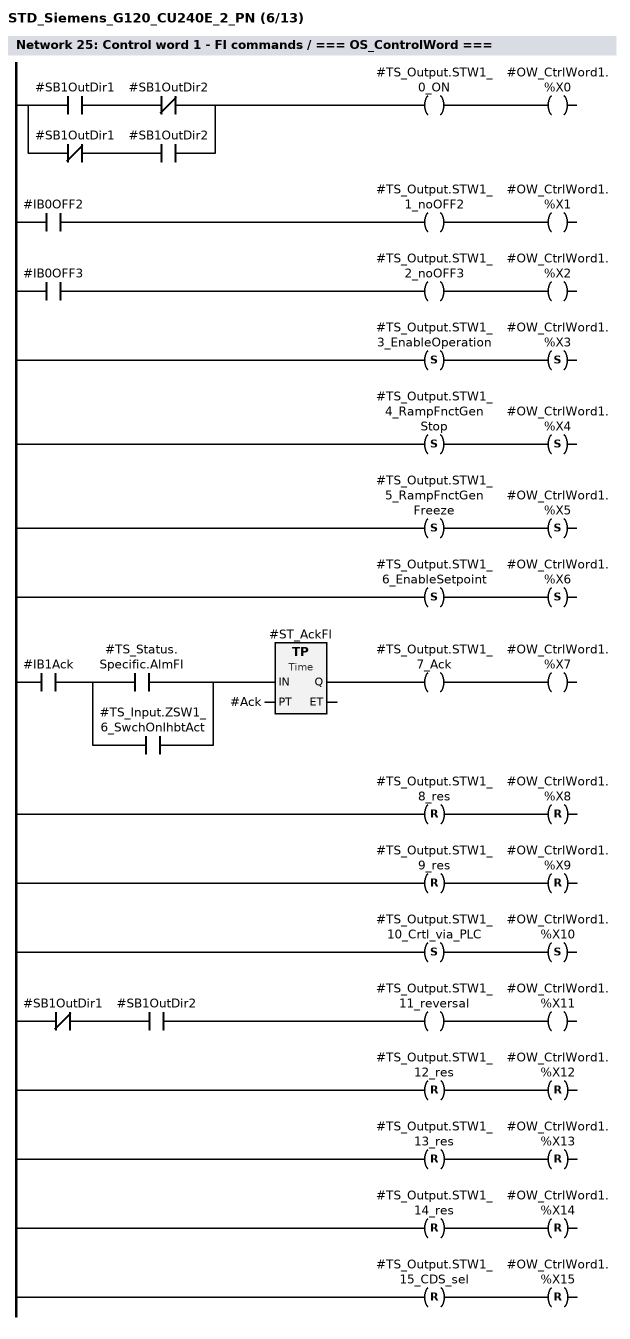
   RUNG wire#powerrail
      Contact( #SB1OutDir1 )
      I_Contact( #SB1OutDir2 )
      wire#w1
      Coil( #TS_Output.STW1_0_ON )
      Coil( #OW_CtrlWord1.%X0 )
   END_RUNG
   RUNG wire#powerrail
      I_Contact( #SB1OutDir1 )
      Contact( #SB1OutDir2 )
   END_RUNG wire#w1
   RUNG wire#powerrail
      Contact( #IB0OFF2 )
      Coil( #TS_Output.STW1_1_noOFF2 )
      Coil( #OW_CtrlWord1.%X1 )
   END_RUNG
   RUNG wire#powerrail
      Contact( #IB0OFF3 )
      Coil( #TS_Output.STW1_2_noOFF3 )
      Coil( #OW_CtrlWord1.%X2 )
   END_RUNG
   RUNG wire#powerrail
      S_Coil( #TS_Output.STW1_3_EnableOperation )
      S_Coil( #OW_CtrlWord1.%X3 )
   END_RUNG
   RUNG wire#powerrail
      S_Coil( #TS_Output.STW1_4_RampFnctGenStop )
      S_Coil( #OW_CtrlWord1.%X4 )
   END_RUNG
   RUNG wire#powerrail
      S_Coil( #TS_Output.STW1_5_RampFnctGenFreeze )
      S_Coil( #OW_CtrlWord1.%X5 )
   END_RUNG
   RUNG wire#powerrail
      S_Coil( #TS_Output.STW1_6_EnableSetpoint )
      S_Coil( #OW_CtrlWord1.%X6 )
   END_RUNG
   RUNG wire#powerrail
      Contact( #IB1Ack )
      wire#w2
      Contact( #TS_Status.Specific.AlmFI )
      wire#w3
      { S7_Templates := "time_type := Time" } #ST_AckFl.TP(pt := #Ack, et =>)
      Coil( #TS_Output.STW1_7_Ack )
      Coil( #OW_CtrlWord1.%X7 )
   END_RUNG
   RUNG wire#w2
      Contact( #TS_Input.ZSW1_6_SwchOnIhbtAct )
   END_RUNG wire#w3
   RUNG wire#powerrail
      R_Coil( #TS_Output.STW1_8_res )
      R_Coil( #OW_CtrlWord1.%X8 )
   END_RUNG
   RUNG wire#powerrail
      R_Coil( #TS_Output.STW1_9_res )
      R_Coil( #OW_CtrlWord1.%X9 )
   END_RUNG
   RUNG wire#powerrail
      S_Coil( #TS_Output.STW1_10_Crtl_via_PLC )
      S_Coil( #OW_CtrlWord1.%X10 )
   END_RUNG
   RUNG wire#powerrail
      I_Contact( #SB1OutDir1 )
      Contact( #SB1OutDir2 )
      Coil( #TS_Output.STW1_11_reversal )
      Coil( #OW_CtrlWord1.%X11 )
   END_RUNG
   RUNG wire#powerrail
      R_Coil( #TS_Output.STW1_12_res )
      R_Coil( #OW_CtrlWord1.%X12 )
   END_RUNG
   RUNG wire#powerrail
      R_Coil( #TS_Output.STW1_13_res )
      R_Coil( #OW_CtrlWord1.%X13 )
   END_RUNG
   RUNG wire#powerrail
      R_Coil( #TS_Output.STW1_14_res )
      R_Coil( #OW_CtrlWord1.%X14 )
   END_RUNG
   RUNG wire#powerrail
      R_Coil( #TS_Output.STW1_15_CDS_sel )
      R_Coil( #OW_CtrlWord1.%X15 )
   END_RUNG
   // the same network as SCL:
   #TS_Output.STW1_0_ON := (#SB1OutDir1 AND NOT #SB1OutDir2) OR (NOT #SB1OutDir1 AND #SB1OutDir2);
   #OW_CtrlWord1.%X0 := #TS_Output.STW1_0_ON;
   #TS_Output.STW1_1_noOFF2 := #IB0OFF2;
   #OW_CtrlWord1.%X1 := #IB0OFF2;
   #TS_Output.STW1_2_noOFF3 := #IB0OFF3;
   #OW_CtrlWord1.%X2 := #IB0OFF3;
   #TS_Output.STW1_3_EnableOperation := TRUE;
   #OW_CtrlWord1.%X3 := TRUE;
   #TS_Output.STW1_4_RampFnctGenStop := TRUE;
   #OW_CtrlWord1.%X4 := TRUE;
   #TS_Output.STW1_5_RampFnctGenFreeze := TRUE;
   #OW_CtrlWord1.%X5 := TRUE;
   #TS_Output.STW1_6_EnableSetpoint := TRUE;
   #OW_CtrlWord1.%X6 := TRUE;
   #ST_AckFl(IN := #IB1Ack AND (#TS_Status.Specific.AlmFI OR #TS_Input.ZSW1_6_SwchOnIhbtAct), PT := #Ack);   // TP
   #TS_Output.STW1_7_Ack := #ST_AckFl.Q;
   #OW_CtrlWord1.%X7 := #ST_AckFl.Q;
   #TS_Output.STW1_8_res := FALSE;
   #OW_CtrlWord1.%X8 := FALSE;
   #TS_Output.STW1_9_res := FALSE;
   #OW_CtrlWord1.%X9 := FALSE;
   #TS_Output.STW1_10_Crtl_via_PLC := TRUE;
   #OW_CtrlWord1.%X10 := TRUE;
   #TS_Output.STW1_11_reversal := NOT #SB1OutDir1 AND #SB1OutDir2;
   #OW_CtrlWord1.%X11 := #TS_Output.STW1_11_reversal;
   #TS_Output.STW1_12_res := FALSE;
   #OW_CtrlWord1.%X12 := FALSE;
   #TS_Output.STW1_13_res := FALSE;
   #OW_CtrlWord1.%X13 := FALSE;
   #TS_Output.STW1_14_res := FALSE;
   #OW_CtrlWord1.%X14 := FALSE;
   #TS_Output.STW1_15_CDS_sel := FALSE;
   #OW_CtrlWord1.%X15 := FALSE;
END_REGION

REGION Network 26: Control word 2 - setpoint / speed / FI Speed + Ramp
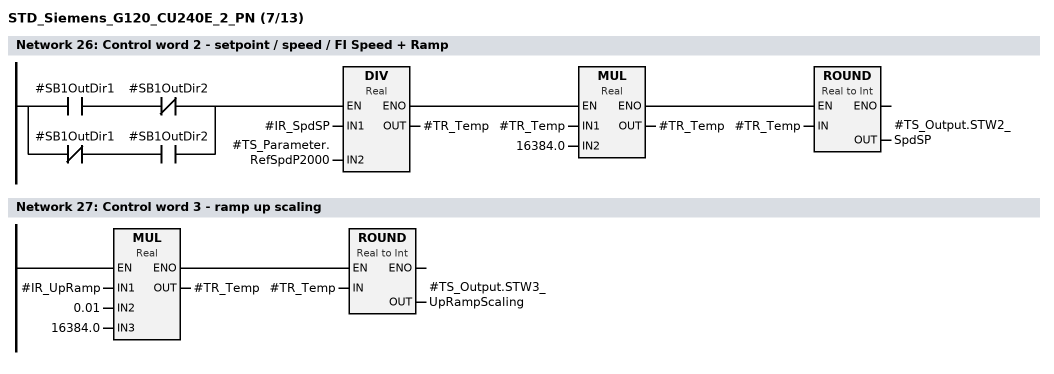
   RUNG wire#powerrail
      Contact( #SB1OutDir1 )
      I_Contact( #SB1OutDir2 )
      wire#w1
      { S7_Templates := "SrcType := Real"; S7_GenerateENO := "TRUE" } Div(in1 := #IR_SpdSP, in2 := #TS_Parameter.RefSpdP2000, out => #TR_Temp)
      { S7_Templates := "SrcType := Real"; S7_GenerateENO := "TRUE" } Mul(in1 := #TR_Temp, in2 := 16384.0, out => #TR_Temp)
      { S7_Templates := "[SrcType := Real, DestType := Int]"; S7_GenerateENO := "TRUE" } Round(in := #TR_Temp, out => #TS_Output.STW2_SpdSP)
   END_RUNG
   RUNG wire#powerrail
      I_Contact( #SB1OutDir1 )
      Contact( #SB1OutDir2 )
   END_RUNG wire#w1
   // the same network as SCL:
   // ENO of a box is taken as its EN; it also drops when the box reports an error
   IF (#SB1OutDir1 AND NOT #SB1OutDir2) OR (NOT #SB1OutDir1 AND #SB1OutDir2) THEN
       #TR_Temp := #IR_SpdSP / #TS_Parameter.RefSpdP2000;
       #TR_Temp := #TR_Temp * 16384.0;
       #TS_Output.STW2_SpdSP := ROUND(#TR_Temp);
   END_IF;
END_REGION

REGION Network 27: Control word 3 - ramp up scaling
   RUNG wire#powerrail
      { S7_Templates := "SrcType := Real"; S7_GenerateENO := "TRUE" } Mul(in1 := #IR_UpRamp, in2 := 0.01, in3 := 16384.0, out => #TR_Temp)
      { S7_Templates := "[SrcType := Real, DestType := Int]"; S7_GenerateENO := "TRUE" } Round(in := #TR_Temp, out => #TS_Output.STW3_UpRampScaling)
   END_RUNG
   // the same network as SCL:
   // ENO of a box is taken as its EN; it also drops when the box reports an error
   #TR_Temp := #IR_UpRamp * 0.01 * 16384.0;
   #TS_Output.STW3_UpRampScaling := ROUND(#TR_Temp);
END_REGION

REGION Network 28: Control word 4 - binary signals
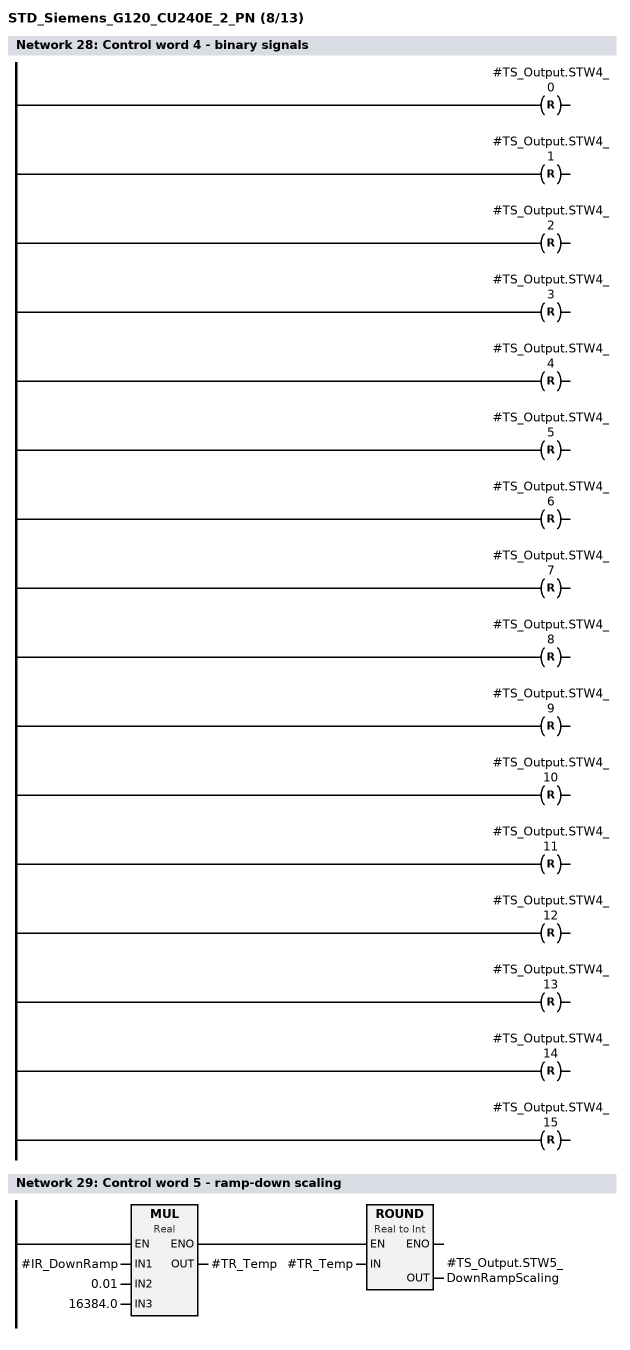
   RUNG wire#powerrail
      R_Coil( #TS_Output.STW4_0 )
   END_RUNG
   RUNG wire#powerrail
      R_Coil( #TS_Output.STW4_1 )
   END_RUNG
   RUNG wire#powerrail
      R_Coil( #TS_Output.STW4_2 )
   END_RUNG
   RUNG wire#powerrail
      R_Coil( #TS_Output.STW4_3 )
   END_RUNG
   RUNG wire#powerrail
      R_Coil( #TS_Output.STW4_4 )
   END_RUNG
   RUNG wire#powerrail
      R_Coil( #TS_Output.STW4_5 )
   END_RUNG
   RUNG wire#powerrail
      R_Coil( #TS_Output.STW4_6 )
   END_RUNG
   RUNG wire#powerrail
      R_Coil( #TS_Output.STW4_7 )
   END_RUNG
   RUNG wire#powerrail
      R_Coil( #TS_Output.STW4_8 )
   END_RUNG
   RUNG wire#powerrail
      R_Coil( #TS_Output.STW4_9 )
   END_RUNG
   RUNG wire#powerrail
      R_Coil( #TS_Output.STW4_10 )
   END_RUNG
   RUNG wire#powerrail
      R_Coil( #TS_Output.STW4_11 )
   END_RUNG
   RUNG wire#powerrail
      R_Coil( #TS_Output.STW4_12 )
   END_RUNG
   RUNG wire#powerrail
      R_Coil( #TS_Output.STW4_13 )
   END_RUNG
   RUNG wire#powerrail
      R_Coil( #TS_Output.STW4_14 )
   END_RUNG
   RUNG wire#powerrail
      R_Coil( #TS_Output.STW4_15 )
   END_RUNG
   // the same network as SCL:
   #TS_Output.STW4_0 := FALSE;
   #TS_Output.STW4_1 := FALSE;
   #TS_Output.STW4_2 := FALSE;
   #TS_Output.STW4_3 := FALSE;
   #TS_Output.STW4_4 := FALSE;
   #TS_Output.STW4_5 := FALSE;
   #TS_Output.STW4_6 := FALSE;
   #TS_Output.STW4_7 := FALSE;
   #TS_Output.STW4_8 := FALSE;
   #TS_Output.STW4_9 := FALSE;
   #TS_Output.STW4_10 := FALSE;
   #TS_Output.STW4_11 := FALSE;
   #TS_Output.STW4_12 := FALSE;
   #TS_Output.STW4_13 := FALSE;
   #TS_Output.STW4_14 := FALSE;
   #TS_Output.STW4_15 := FALSE;
END_REGION

REGION Network 29: Control word 5 - ramp-down scaling
   RUNG wire#powerrail
      { S7_Templates := "SrcType := Real"; S7_GenerateENO := "TRUE" } Mul(in1 := #IR_DownRamp, in2 := 0.01, in3 := 16384.0, out => #TR_Temp)
      { S7_Templates := "[SrcType := Real, DestType := Int]"; S7_GenerateENO := "TRUE" } Round(in := #TR_Temp, out => #TS_Output.STW5_DownRampScaling)
   END_RUNG
   // the same network as SCL:
   // ENO of a box is taken as its EN; it also drops when the box reports an error
   #TR_Temp := #IR_DownRamp * 0.01 * 16384.0;
   #TS_Output.STW5_DownRampScaling := ROUND(#TR_Temp);
END_REGION

REGION Network 30: Control word 6 - reserve
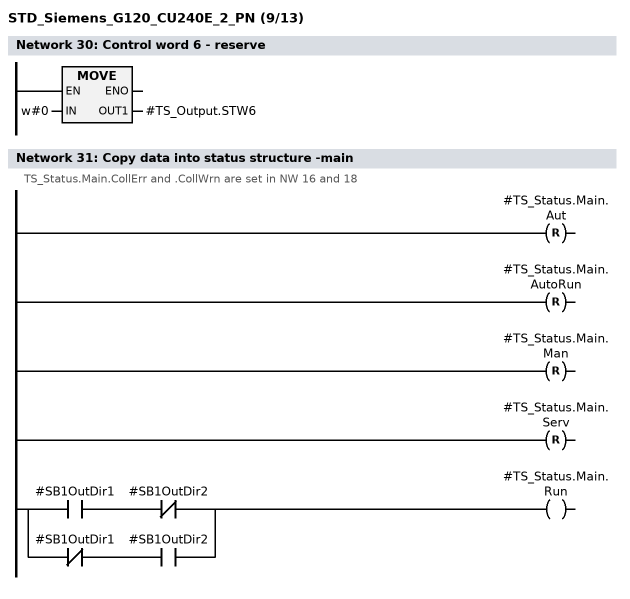
   RUNG wire#powerrail
      { S7_GenerateENO := "TRUE" } Move(in := w#0, out1 => #TS_Output.STW6)
   END_RUNG
   // the same network as SCL:
   #TS_Output.STW6 := w#0;
END_REGION

REGION Network 31: Copy data into status structure -main
   // TS_Status.Main.CollErr and .CollWrn are set in NW 16 and 18
   RUNG wire#powerrail
      R_Coil( #TS_Status.Main.Aut )
   END_RUNG
   RUNG wire#powerrail
      R_Coil( #TS_Status.Main.AutoRun )
   END_RUNG
   RUNG wire#powerrail
      R_Coil( #TS_Status.Main.Man )
   END_RUNG
   RUNG wire#powerrail
      R_Coil( #TS_Status.Main.Serv )
   END_RUNG
   RUNG wire#powerrail
      Contact( #SB1OutDir1 )
      I_Contact( #SB1OutDir2 )
      wire#w1
      Coil( #TS_Status.Main.Run )
   END_RUNG
   RUNG wire#powerrail
      I_Contact( #SB1OutDir1 )
      Contact( #SB1OutDir2 )
   END_RUNG wire#w1
   // the same network as SCL:
   #TS_Status.Main.Aut := FALSE;
   #TS_Status.Main.AutoRun := FALSE;
   #TS_Status.Main.Man := FALSE;
   #TS_Status.Main.Serv := FALSE;
   #TS_Status.Main.Run := (#SB1OutDir1 AND NOT #SB1OutDir2) OR (NOT #SB1OutDir1 AND #SB1OutDir2);
END_REGION

REGION Network 32: Copy data into status structure- specific
   // TS_Status.Specific.AlmFI and .AlmM1 and .AlmCtrl are set in NW 16
   // TS_Status.Specific.Rel is set in NW 22
   // TS_Status.Specific.Spd and .Curr and .Trq are set in NW 19 and 20 and 21
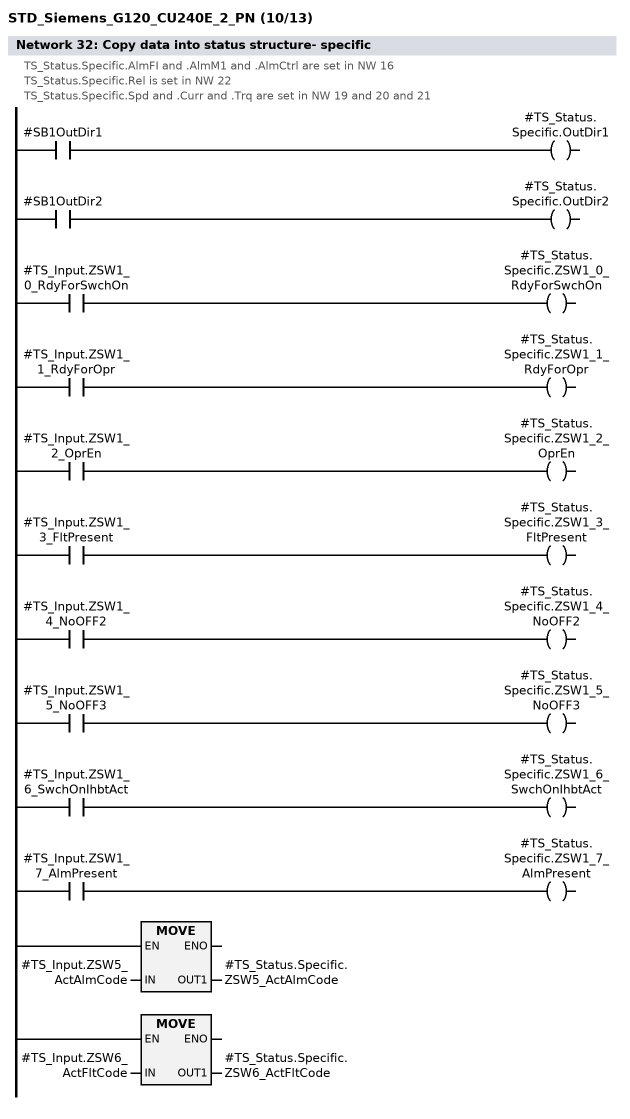
   RUNG wire#powerrail
      Contact( #SB1OutDir1 )
      Coil( #TS_Status.Specific.OutDir1 )
   END_RUNG
   RUNG wire#powerrail
      Contact( #SB1OutDir2 )
      Coil( #TS_Status.Specific.OutDir2 )
   END_RUNG
   RUNG wire#powerrail
      Contact( #TS_Input.ZSW1_0_RdyForSwchOn )
      Coil( #TS_Status.Specific.ZSW1_0_RdyForSwchOn )
   END_RUNG
   RUNG wire#powerrail
      Contact( #TS_Input.ZSW1_1_RdyForOpr )
      Coil( #TS_Status.Specific.ZSW1_1_RdyForOpr )
   END_RUNG
   RUNG wire#powerrail
      Contact( #TS_Input.ZSW1_2_OprEn )
      Coil( #TS_Status.Specific.ZSW1_2_OprEn )
   END_RUNG
   RUNG wire#powerrail
      Contact( #TS_Input.ZSW1_3_FltPresent )
      Coil( #TS_Status.Specific.ZSW1_3_FltPresent )
   END_RUNG
   RUNG wire#powerrail
      Contact( #TS_Input.ZSW1_4_NoOFF2 )
      Coil( #TS_Status.Specific.ZSW1_4_NoOFF2 )
   END_RUNG
   RUNG wire#powerrail
      Contact( #TS_Input.ZSW1_5_NoOFF3 )
      Coil( #TS_Status.Specific.ZSW1_5_NoOFF3 )
   END_RUNG
   RUNG wire#powerrail
      Contact( #TS_Input.ZSW1_6_SwchOnIhbtAct )
      Coil( #TS_Status.Specific.ZSW1_6_SwchOnIhbtAct )
   END_RUNG
   RUNG wire#powerrail
      Contact( #TS_Input.ZSW1_7_AlmPresent )
      Coil( #TS_Status.Specific.ZSW1_7_AlmPresent )
   END_RUNG
   RUNG wire#powerrail
      { S7_GenerateENO := "TRUE" } Move(in := #TS_Input.ZSW5_ActAlmCode, out1 => #TS_Status.Specific.ZSW5_ActAlmCode)
   END_RUNG
   RUNG wire#powerrail
      { S7_GenerateENO := "TRUE" } Move(in := #TS_Input.ZSW6_ActFltCode, out1 => #TS_Status.Specific.ZSW6_ActFltCode)
   END_RUNG
   // the same network as SCL:
   #TS_Status.Specific.OutDir1 := #SB1OutDir1;
   #TS_Status.Specific.OutDir2 := #SB1OutDir2;
   #TS_Status.Specific.ZSW1_0_RdyForSwchOn := #TS_Input.ZSW1_0_RdyForSwchOn;
   #TS_Status.Specific.ZSW1_1_RdyForOpr := #TS_Input.ZSW1_1_RdyForOpr;
   #TS_Status.Specific.ZSW1_2_OprEn := #TS_Input.ZSW1_2_OprEn;
   #TS_Status.Specific.ZSW1_3_FltPresent := #TS_Input.ZSW1_3_FltPresent;
   #TS_Status.Specific.ZSW1_4_NoOFF2 := #TS_Input.ZSW1_4_NoOFF2;
   #TS_Status.Specific.ZSW1_5_NoOFF3 := #TS_Input.ZSW1_5_NoOFF3;
   #TS_Status.Specific.ZSW1_6_SwchOnIhbtAct := #TS_Input.ZSW1_6_SwchOnIhbtAct;
   #TS_Status.Specific.ZSW1_7_AlmPresent := #TS_Input.ZSW1_7_AlmPresent;
   #TS_Status.Specific.ZSW5_ActAlmCode := #TS_Input.ZSW5_ActAlmCode;
   #TS_Status.Specific.ZSW6_ActFltCode := #TS_Input.ZSW6_ActFltCode;
END_REGION

REGION Network 33: Clear TS_Command
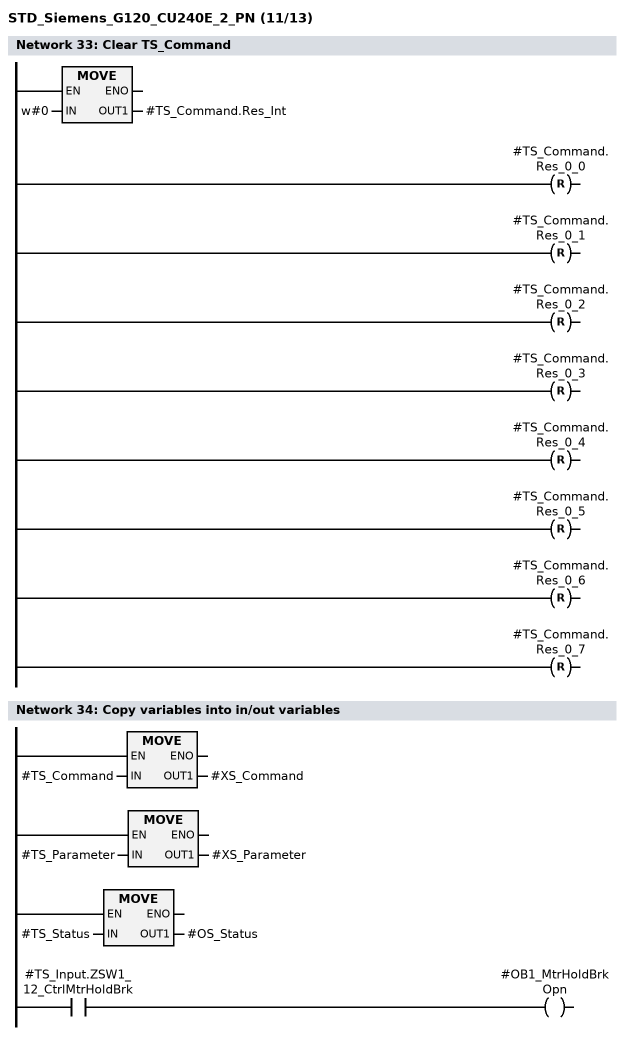
   RUNG wire#powerrail
      { S7_GenerateENO := "TRUE" } Move(in := w#0, out1 => #TS_Command.Res_Int)
   END_RUNG
   RUNG wire#powerrail
      R_Coil( #TS_Command.Res_0_0 )
   END_RUNG
   RUNG wire#powerrail
      R_Coil( #TS_Command.Res_0_1 )
   END_RUNG
   RUNG wire#powerrail
      R_Coil( #TS_Command.Res_0_2 )
   END_RUNG
   RUNG wire#powerrail
      R_Coil( #TS_Command.Res_0_3 )
   END_RUNG
   RUNG wire#powerrail
      R_Coil( #TS_Command.Res_0_4 )
   END_RUNG
   RUNG wire#powerrail
      R_Coil( #TS_Command.Res_0_5 )
   END_RUNG
   RUNG wire#powerrail
      R_Coil( #TS_Command.Res_0_6 )
   END_RUNG
   RUNG wire#powerrail
      R_Coil( #TS_Command.Res_0_7 )
   END_RUNG
   // the same network as SCL:
   #TS_Command.Res_Int := w#0;
   #TS_Command.Res_0_0 := FALSE;
   #TS_Command.Res_0_1 := FALSE;
   #TS_Command.Res_0_2 := FALSE;
   #TS_Command.Res_0_3 := FALSE;
   #TS_Command.Res_0_4 := FALSE;
   #TS_Command.Res_0_5 := FALSE;
   #TS_Command.Res_0_6 := FALSE;
   #TS_Command.Res_0_7 := FALSE;
END_REGION

REGION Network 34: Copy variables into in/out variables
   RUNG wire#powerrail
      { S7_GenerateENO := "TRUE" } Move(in := #TS_Command, out1 => #XS_Command)
   END_RUNG
   RUNG wire#powerrail
      { S7_GenerateENO := "TRUE" } Move(in := #TS_Parameter, out1 => #XS_Parameter)
   END_RUNG
   RUNG wire#powerrail
      { S7_GenerateENO := "TRUE" } Move(in := #TS_Status, out1 => #OS_Status)
   END_RUNG
   RUNG wire#powerrail
      Contact( #TS_Input.ZSW1_12_CtrlMtrHoldBrk )
      Coil( #OB1_MtrHoldBrkOpn )
   END_RUNG
   // the same network as SCL:
   #XS_Command := #TS_Command;
   #XS_Parameter := #TS_Parameter;
   #OS_Status := #TS_Status;
   #OB1_MtrHoldBrkOpn := #TS_Input.ZSW1_12_CtrlMtrHoldBrk;
END_REGION

REGION Network 35: Copy alarms into status - error
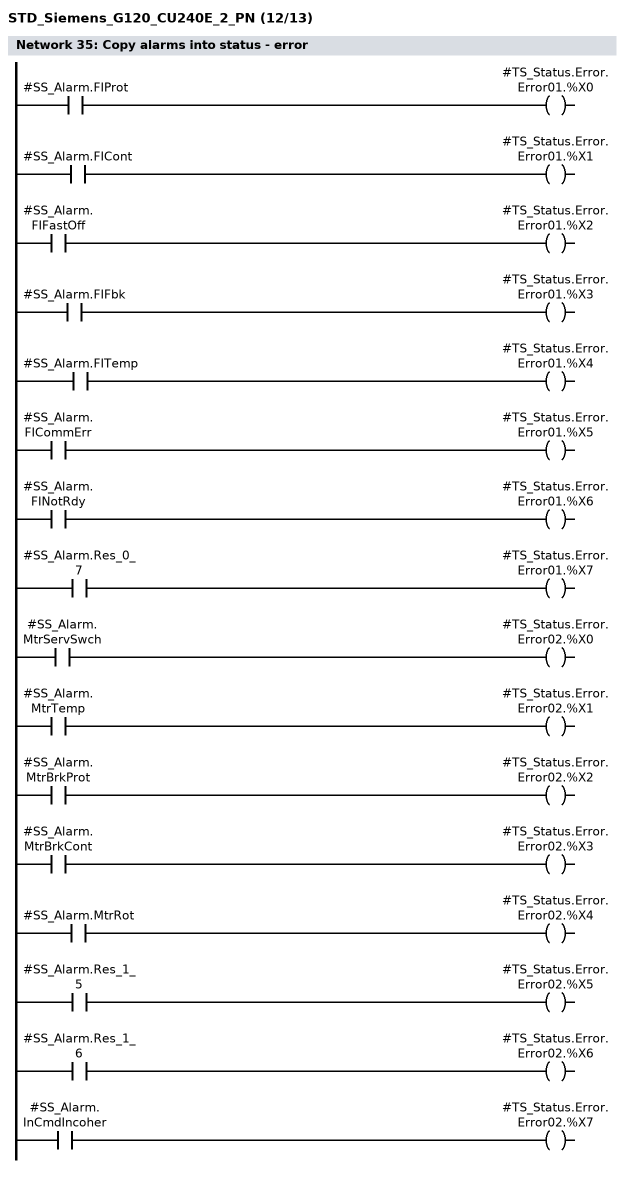
   RUNG wire#powerrail
      Contact( #SS_Alarm.FIProt )
      Coil( #TS_Status.Error.Error01.%X0 )
   END_RUNG
   RUNG wire#powerrail
      Contact( #SS_Alarm.FICont )
      Coil( #TS_Status.Error.Error01.%X1 )
   END_RUNG
   RUNG wire#powerrail
      Contact( #SS_Alarm.FIFastOff )
      Coil( #TS_Status.Error.Error01.%X2 )
   END_RUNG
   RUNG wire#powerrail
      Contact( #SS_Alarm.FIFbk )
      Coil( #TS_Status.Error.Error01.%X3 )
   END_RUNG
   RUNG wire#powerrail
      Contact( #SS_Alarm.FITemp )
      Coil( #TS_Status.Error.Error01.%X4 )
   END_RUNG
   RUNG wire#powerrail
      Contact( #SS_Alarm.FICommErr )
      Coil( #TS_Status.Error.Error01.%X5 )
   END_RUNG
   RUNG wire#powerrail
      Contact( #SS_Alarm.FINotRdy )
      Coil( #TS_Status.Error.Error01.%X6 )
   END_RUNG
   RUNG wire#powerrail
      Contact( #SS_Alarm.Res_0_7 )
      Coil( #TS_Status.Error.Error01.%X7 )
   END_RUNG
   RUNG wire#powerrail
      Contact( #SS_Alarm.MtrServSwch )
      Coil( #TS_Status.Error.Error02.%X0 )
   END_RUNG
   RUNG wire#powerrail
      Contact( #SS_Alarm.MtrTemp )
      Coil( #TS_Status.Error.Error02.%X1 )
   END_RUNG
   RUNG wire#powerrail
      Contact( #SS_Alarm.MtrBrkProt )
      Coil( #TS_Status.Error.Error02.%X2 )
   END_RUNG
   RUNG wire#powerrail
      Contact( #SS_Alarm.MtrBrkCont )
      Coil( #TS_Status.Error.Error02.%X3 )
   END_RUNG
   RUNG wire#powerrail
      Contact( #SS_Alarm.MtrRot )
      Coil( #TS_Status.Error.Error02.%X4 )
   END_RUNG
   RUNG wire#powerrail
      Contact( #SS_Alarm.Res_1_5 )
      Coil( #TS_Status.Error.Error02.%X5 )
   END_RUNG
   RUNG wire#powerrail
      Contact( #SS_Alarm.Res_1_6 )
      Coil( #TS_Status.Error.Error02.%X6 )
   END_RUNG
   RUNG wire#powerrail
      Contact( #SS_Alarm.InCmdIncoher )
      Coil( #TS_Status.Error.Error02.%X7 )
   END_RUNG
   // the same network as SCL:
   #TS_Status.Error.Error01.%X0 := #SS_Alarm.FIProt;
   #TS_Status.Error.Error01.%X1 := #SS_Alarm.FICont;
   #TS_Status.Error.Error01.%X2 := #SS_Alarm.FIFastOff;
   #TS_Status.Error.Error01.%X3 := #SS_Alarm.FIFbk;
   #TS_Status.Error.Error01.%X4 := #SS_Alarm.FITemp;
   #TS_Status.Error.Error01.%X5 := #SS_Alarm.FICommErr;
   #TS_Status.Error.Error01.%X6 := #SS_Alarm.FINotRdy;
   #TS_Status.Error.Error01.%X7 := #SS_Alarm.Res_0_7;
   #TS_Status.Error.Error02.%X0 := #SS_Alarm.MtrServSwch;
   #TS_Status.Error.Error02.%X1 := #SS_Alarm.MtrTemp;
   #TS_Status.Error.Error02.%X2 := #SS_Alarm.MtrBrkProt;
   #TS_Status.Error.Error02.%X3 := #SS_Alarm.MtrBrkCont;
   #TS_Status.Error.Error02.%X4 := #SS_Alarm.MtrRot;
   #TS_Status.Error.Error02.%X5 := #SS_Alarm.Res_1_5;
   #TS_Status.Error.Error02.%X6 := #SS_Alarm.Res_1_6;
   #TS_Status.Error.Error02.%X7 := #SS_Alarm.InCmdIncoher;
END_REGION

REGION Network 36: Copy warnings into status - error
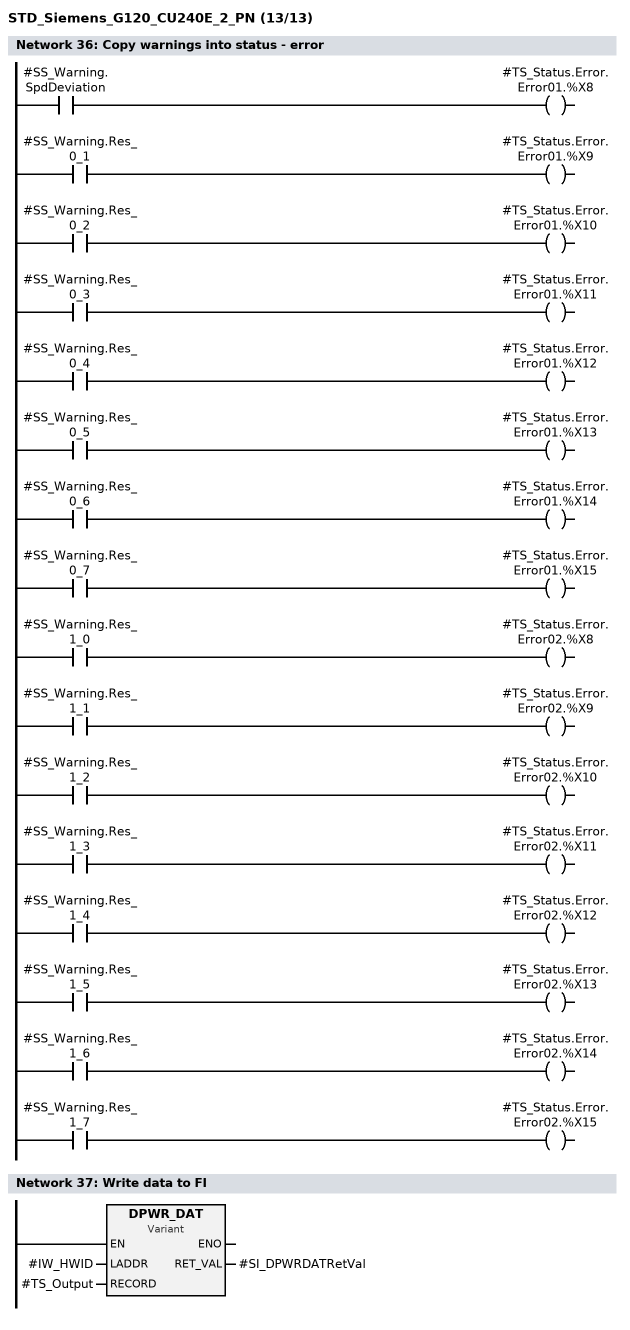
   RUNG wire#powerrail
      Contact( #SS_Warning.SpdDeviation )
      Coil( #TS_Status.Error.Error01.%X8 )
   END_RUNG
   RUNG wire#powerrail
      Contact( #SS_Warning.Res_0_1 )
      Coil( #TS_Status.Error.Error01.%X9 )
   END_RUNG
   RUNG wire#powerrail
      Contact( #SS_Warning.Res_0_2 )
      Coil( #TS_Status.Error.Error01.%X10 )
   END_RUNG
   RUNG wire#powerrail
      Contact( #SS_Warning.Res_0_3 )
      Coil( #TS_Status.Error.Error01.%X11 )
   END_RUNG
   RUNG wire#powerrail
      Contact( #SS_Warning.Res_0_4 )
      Coil( #TS_Status.Error.Error01.%X12 )
   END_RUNG
   RUNG wire#powerrail
      Contact( #SS_Warning.Res_0_5 )
      Coil( #TS_Status.Error.Error01.%X13 )
   END_RUNG
   RUNG wire#powerrail
      Contact( #SS_Warning.Res_0_6 )
      Coil( #TS_Status.Error.Error01.%X14 )
   END_RUNG
   RUNG wire#powerrail
      Contact( #SS_Warning.Res_0_7 )
      Coil( #TS_Status.Error.Error01.%X15 )
   END_RUNG
   RUNG wire#powerrail
      Contact( #SS_Warning.Res_1_0 )
      Coil( #TS_Status.Error.Error02.%X8 )
   END_RUNG
   RUNG wire#powerrail
      Contact( #SS_Warning.Res_1_1 )
      Coil( #TS_Status.Error.Error02.%X9 )
   END_RUNG
   RUNG wire#powerrail
      Contact( #SS_Warning.Res_1_2 )
      Coil( #TS_Status.Error.Error02.%X10 )
   END_RUNG
   RUNG wire#powerrail
      Contact( #SS_Warning.Res_1_3 )
      Coil( #TS_Status.Error.Error02.%X11 )
   END_RUNG
   RUNG wire#powerrail
      Contact( #SS_Warning.Res_1_4 )
      Coil( #TS_Status.Error.Error02.%X12 )
   END_RUNG
   RUNG wire#powerrail
      Contact( #SS_Warning.Res_1_5 )
      Coil( #TS_Status.Error.Error02.%X13 )
   END_RUNG
   RUNG wire#powerrail
      Contact( #SS_Warning.Res_1_6 )
      Coil( #TS_Status.Error.Error02.%X14 )
   END_RUNG
   RUNG wire#powerrail
      Contact( #SS_Warning.Res_1_7 )
      Coil( #TS_Status.Error.Error02.%X15 )
   END_RUNG
   // the same network as SCL:
   #TS_Status.Error.Error01.%X8 := #SS_Warning.SpdDeviation;
   #TS_Status.Error.Error01.%X9 := #SS_Warning.Res_0_1;
   #TS_Status.Error.Error01.%X10 := #SS_Warning.Res_0_2;
   #TS_Status.Error.Error01.%X11 := #SS_Warning.Res_0_3;
   #TS_Status.Error.Error01.%X12 := #SS_Warning.Res_0_4;
   #TS_Status.Error.Error01.%X13 := #SS_Warning.Res_0_5;
   #TS_Status.Error.Error01.%X14 := #SS_Warning.Res_0_6;
   #TS_Status.Error.Error01.%X15 := #SS_Warning.Res_0_7;
   #TS_Status.Error.Error02.%X8 := #SS_Warning.Res_1_0;
   #TS_Status.Error.Error02.%X9 := #SS_Warning.Res_1_1;
   #TS_Status.Error.Error02.%X10 := #SS_Warning.Res_1_2;
   #TS_Status.Error.Error02.%X11 := #SS_Warning.Res_1_3;
   #TS_Status.Error.Error02.%X12 := #SS_Warning.Res_1_4;
   #TS_Status.Error.Error02.%X13 := #SS_Warning.Res_1_5;
   #TS_Status.Error.Error02.%X14 := #SS_Warning.Res_1_6;
   #TS_Status.Error.Error02.%X15 := #SS_Warning.Res_1_7;
END_REGION

REGION Network 37: Write data to FI
   RUNG wire#powerrail
      { S7_Templates := "[ptr_type := Variant, laddr_type := HW_IO]" } DPWR_DAT(LADDR := #IW_HWID, RECORD := #TS_Output, RET_VAL => #SI_DPWRDATRetVal)
   END_RUNG
   // the same network as SCL:
   #SI_DPWRDATRetVal := DPWR_DAT(LADDR := #IW_HWID, RECORD := #TS_Output);
END_REGION
END_FUNCTION_BLOCK
